# B&R Automation Studio project Ampel
Automation Studio 6.3.2.2; Traffic Ligh in B&R 6.3; technology packages: mappView 6.0.0, OpcUaCs 6.0.0

## Configuration Config1

CPU PC_any, AutomationRuntime 6.3.0, Build 11.3.0, Vc 6.0.0

### Hardware
```
PC : PC_any v1.1.2.0 (OrderNumber=PC)
  ConfigurationID = Ampel_Config1
  FileDevice1
  FileDeviceName1 = USER
  FileDevicePath1 = USER_PATH
```

## Logical view

### Program Logical/Ampel (ANSIC)

#### Main.cpp - Init, cyclic, exit code
```cpp
#include <bur/plctypes.h>

#ifdef _DEFAULT_INCLUDES
#include <AsDefault.h>
#endif

// amount of memory to be allocated for heap storage must be specified
// for every ANSI C++ program with the bur_heap_size variable
unsigned long bur_heap_size = 0xFFFF;

#include "machine.hpp"
#include "Logging.hpp"
#include "States.hpp"

////////////////////////////////////////////////////////////////////////////////

// shared data storage instance
Context context;
FSM::Instance machine{context};

void _INIT ProgramInit(void)
{
	// Insert code here
	CyclesCount = 0;
	ClearTraceLog();
	DurationRed = 5;
	DurationYellow = 3;
	DurationGreen = 5;
	DurationGreenBlinking = 3;
	LightRed = false;
	LightYellow = false;
	LightGreen = false;
	CountDownRedON = false;
	CountDownGreenON = false;
}

void _CYCLIC ProgramCyclic(void)
{
	// Insert code here
	machine.update();
	LightRedOFF = !LightRed; LightYellowOFF = !LightYellow; LightGreenOFF = !LightGreen;
	CountDownRedON = LightRed;
	CyclesCount++;
	TraceMessage("---cycle---");
}

void _EXIT ProgramExit(void)
{
	// Insert code here
}
```

#### Variables.var - Local variables
```iecst
VAR
	DurationGreenBlinking : USINT;
	DurationGreen : USINT;
	DurationYellow : USINT;
	DurationRed : USINT;
	LightYellow : BOOL;
	LightRed : BOOL;
	LightGreen : BOOL;
	CyclesCount : USINT;
	TraceMessages : ARRAY[0..200] OF STRING[80];
	LightYellowOFF : BOOL;
	CountDown : USINT;
	LightRedOFF : BOOL;
	LightGreenOFF : BOOL;
	CountDownRedON : BOOL;
	CountDownGreenON : BOOL;
END_VAR

VAR CONSTANT

END_VAR
```

#### machine.hpp
```cpp
// https://github.com/andrew-gresyk/HFSM2
// include/hfsm2/machine.hpp
// HFSM2 (hierarchical state machine for games and interactive applications)
// 2.8.0 (2025-07-20)
//
// Created by Andrew Gresyk
//
// Licensed under the MIT License;
// you may not use this file except in compliance with the License.
//
//
// MIT License
//
// Copyright (c) 2025
//
// Permission is hereby granted, free of charge, to any person obtaining a copy
// of this software and associated documentation files (the "Software"), to deal
// in the Software without restriction, including without limitation the rights
// to use, copy, modify, merge, publish, distribute, sublicense, and/or sell
// copies of the Software, and to permit persons to whom the Software is
// furnished to do so, subject to the following conditions:
//
// The above copyright notice and this permission notice shall be included in all
// copies or substantial portions of the Software.
//
// THE SOFTWARE IS PROVIDED "AS IS", WITHOUT WARRANTY OF ANY KIND, EXPRESS OR
// IMPLIED, INCLUDING BUT NOT LIMITED TO THE WARRANTIES OF MERCHANTABILITY,
// FITNESS FOR A PARTICULAR PURPOSE AND NONINFRINGEMENT. IN NO EVENT SHALL THE
// AUTHORS OR COPYRIGHT HOLDERS BE LIABLE FOR ANY CLAIM, DAMAGES OR OTHER
// LIABILITY, WHETHER IN AN ACTION OF CONTRACT, TORT OR OTHERWISE, ARISING FROM,
// OUT OF OR IN CONNECTION WITH THE SOFTWARE OR THE USE OR OTHER DEALINGS IN THE
// SOFTWARE.

#pragma once

#define HFSM2_VERSION_MAJOR 2
#define HFSM2_VERSION_MINOR 8
#define HFSM2_VERSION_PATCH 0

#define HFSM2_VERSION (10000 * HFSM2_VERSION_MAJOR + 100 * HFSM2_VERSION_MINOR + HFSM2_VERSION_PATCH)

#include <stdint.h>			// uint32_t, uint64_t
#include <string.h>			// memcpy_s()

#include <new>
#ifndef HFSM2_DISABLE_TYPEINDEX
#include <typeindex>
#endif

#if defined _DEBUG && _MSC_VER
#include <intrin.h>		// __debugbreak()
#endif

#define HFSM2_UNUSED(x)

#define HFSM2_ATTRIBUTE(A)								   HFSM2_ATTRIBUTE_##A()

#ifndef __has_cpp_attribute
#define __has_cpp_attribute(x)											   0
#endif

#if __has_cpp_attribute(fallthrough)
#define HFSM2_ATTRIBUTE_FALLTHROUGH()						 [[fallthrough]]
#elif __has_cpp_attribute(clang::fallthrough)
#define HFSM2_ATTRIBUTE_FALLTHROUGH()				  [[clang::fallthrough]]
#elif __has_cpp_attribute(gnu::fallthrough)
#define HFSM2_ATTRIBUTE_FALLTHROUGH()					[[gnu::fallthrough]]
#else
#define HFSM2_ATTRIBUTE_FALLTHROUGH()
#endif

#if __has_cpp_attribute(no_unique_address)
#define HFSM2_ATTRIBUTE_NO_UNIQUE_ADDRESS()			   [[no_unique_address]]
#else
#define HFSM2_ATTRIBUTE_NO_UNIQUE_ADDRESS()
#endif

#define HFSM2_CONSTEXPR(A)								   HFSM2_CONSTEXPR_##A()

#define HFSM2_CONSTEXPR_NO()

#define HFSM2_CONSTEXPR_11()										   constexpr

#if __cplusplus >= 201402L
#define HFSM2_CONSTEXPR_14()									   constexpr
#else
#define HFSM2_CONSTEXPR_14()										  inline
#endif

#if __cplusplus >= 201703L
#define HFSM2_CONSTEXPR_17()									   constexpr
#else
#define HFSM2_CONSTEXPR_17()										  inline
#endif

#if __cplusplus >= 202002L
#define HFSM2_CONSTEXPR_20()									   constexpr
#else
#define HFSM2_CONSTEXPR_20()										  inline
#endif

#if defined _MSC_VER
#define HFSM2_EMPTY_BASES							 __declspec(empty_bases)
#else
#define HFSM2_EMPTY_BASES
#endif

#define HFSM2_ARCHITECTURE(A)							HFSM2_ARCHITECTURE_##A()

#if INTPTR_MAX == INT64_MAX
#define HFSM2_ARCHITECTURE_64BIT()										true
#define HFSM2_ARCHITECTURE_32BIT()									   false

#define HFSM2_64BIT_OR_32BIT(p64, p32)									 p64
#elif INTPTR_MAX == INT32_MAX
#define HFSM2_ARCHITECTURE_64BIT()									   false
#define HFSM2_ARCHITECTURE_32BIT()										true

#define HFSM2_64BIT_OR_32BIT(p64, p32)									 p32
#else
#error
#endif

#if defined _DEBUG && defined _MSC_VER
#define HFSM2_BREAK()										  __debugbreak()
#define HFSM2_BREAK_AVAILABLE()											true
#else
#define HFSM2_BREAK()											  ((void) 0)
#define HFSM2_BREAK_AVAILABLE()										   false
#endif

#ifdef _DEBUG
#define HFSM2_IF_DEBUG(...)										 __VA_ARGS__
#define HFSM2_UNLESS_DEBUG(...)
#define HFSM2_DEBUG_OR(y, n)											   y
#else
#define HFSM2_IF_DEBUG(...)
#define HFSM2_UNLESS_DEBUG(...)									 __VA_ARGS__
#define HFSM2_DEBUG_OR(y, n)											   n
#endif

#if HFSM2_BREAK_AVAILABLE() && defined HFSM2_ENABLE_ASSERT
#define HFSM2_ASSERT_AVAILABLE()										true
#define HFSM2_IF_ASSERT(...)									 __VA_ARGS__
#define HFSM2_CHECKED(x)					   (!!(x) || (HFSM2_BREAK(), 0))
#define HFSM2_ASSERT(x)						   (!!(x) || (HFSM2_BREAK(), 0))
#define HFSM2_ASSERT_OR(y, n)											   y
#else
#define HFSM2_ASSERT_AVAILABLE()									   false
#define HFSM2_IF_ASSERT(...)
#define HFSM2_CHECKED(x)												   x
#define HFSM2_ASSERT(x)											  ((void) 0)
#define HFSM2_ASSERT_OR(y, n)											   n
#endif

#if defined _MSC_VER || defined __clang_major__ && __clang_major__ >= 7
#define HFSM2_EXPLICIT_MEMBER_SPECIALIZATION_AVAILABLE()				true
#else
#define HFSM2_EXPLICIT_MEMBER_SPECIALIZATION_AVAILABLE()			   false
#endif

#ifdef HFSM2_ENABLE_ALL
#define HFSM2_ENABLE_DEBUG_STATE_TYPE
#define HFSM2_ENABLE_PLANS
#define HFSM2_ENABLE_SERIALIZATION
#define HFSM2_ENABLE_STRUCTURE_REPORT
#define HFSM2_ENABLE_TRANSITION_HISTORY
#define HFSM2_ENABLE_UTILITY_THEORY
#endif

#ifndef HFSM2_DISABLE_TYPEINDEX
#define HFSM2_TYPEINDEX_AVAILABLE()										true
#define HFSM2_IF_TYPEINDEX(...)									 __VA_ARGS__
#define HFSM2_TYPEINDEX_MASK										(1 << 0)
#else
#define HFSM2_TYPEINDEX_AVAILABLE()									   false
#define HFSM2_IF_TYPEINDEX(...)
#define HFSM2_TYPEINDEX_MASK										(0 << 0)
#endif

#ifdef HFSM2_ENABLE_DEBUG_STATE_TYPE
#define HFSM2_DEBUG_STATE_TYPE_AVAILABLE()								true
#define HFSM2_DEBUG_STATE_TYPE_MASK									(1 << 1)
#else
#define HFSM2_DEBUG_STATE_TYPE_AVAILABLE()							   false
#define HFSM2_DEBUG_STATE_TYPE_MASK									(0 << 1)
#endif

#ifdef HFSM2_ENABLE_PLANS
#define HFSM2_PLANS_AVAILABLE()											true
#define HFSM2_IF_PLANS(...)										 __VA_ARGS__
#define HFSM2_PLANS_MASK											(1 << 2)
#else
#define HFSM2_PLANS_AVAILABLE()										   false
#define HFSM2_IF_PLANS(...)
#define HFSM2_PLANS_MASK											(0 << 2)
#endif

#ifdef HFSM2_ENABLE_SERIALIZATION
#define HFSM2_SERIALIZATION_AVAILABLE()									true
#define HFSM2_IF_SERIALIZATION(...)								 __VA_ARGS__
#define HFSM2_SERIALIZATION_MASK									(1 << 3)
#else
#define HFSM2_SERIALIZATION_AVAILABLE()								   false
#define HFSM2_IF_SERIALIZATION(...)
#define HFSM2_SERIALIZATION_MASK									(0 << 3)
#endif

#ifdef HFSM2_ENABLE_STRUCTURE_REPORT
#define HFSM2_STRUCTURE_REPORT_AVAILABLE()								true
#define HFSM2_IF_STRUCTURE_REPORT(...)							 __VA_ARGS__
#define HFSM2_STRUCTURE_REPORT_MASK									(1 << 4)
#else
#define HFSM2_STRUCTURE_REPORT_AVAILABLE()							   false
#define HFSM2_IF_STRUCTURE_REPORT(...)
#define HFSM2_STRUCTURE_REPORT_MASK									(0 << 4)
#endif

#ifdef HFSM2_ENABLE_TRANSITION_HISTORY
#define HFSM2_TRANSITION_HISTORY_AVAILABLE()							true
#define HFSM2_IF_TRANSITION_HISTORY(...)						 __VA_ARGS__
#define HFSM2_TRANSITION_HISTORY_MASK								(1 << 5)
#else
#define HFSM2_TRANSITION_HISTORY_AVAILABLE()						   false
#define HFSM2_IF_TRANSITION_HISTORY(...)
#define HFSM2_TRANSITION_HISTORY_MASK								(0 << 5)
#endif

#ifdef HFSM2_ENABLE_UTILITY_THEORY
#define HFSM2_UTILITY_THEORY_AVAILABLE()								true
#define HFSM2_IF_UTILITY_THEORY(...)							 __VA_ARGS__
#define HFSM2_UTILITY_THEORY_MASK									(1 << 6)
#else
#define HFSM2_UTILITY_THEORY_AVAILABLE()							   false
#define HFSM2_IF_UTILITY_THEORY(...)
#define HFSM2_UTILITY_THEORY_MASK									(0 << 6)
#endif

#ifdef HFSM2_ENABLE_VERBOSE_DEBUG_LOG
#define HFSM2_ENABLE_LOG_INTERFACE

#define HFSM2_VERBOSE_DEBUG_LOG_AVAILABLE()								true
#define HFSM2_VERBOSE_DEBUG_LOG_MASK								(1 << 7)
#else
#define HFSM2_VERBOSE_DEBUG_LOG_AVAILABLE()							   false
#define HFSM2_VERBOSE_DEBUG_LOG_MASK								(0 << 7)
#endif

#ifdef HFSM2_ENABLE_LOG_INTERFACE
#define HFSM2_LOG_INTERFACE_AVAILABLE()									true
#define HFSM2_IF_LOG_INTERFACE(...)								 __VA_ARGS__
#define HFSM2_LOG_INTERFACE_MASK									(1 << 8)

#define HFSM2_LOG_TRANSITION(CONTEXT, ORIGIN, TYPE, DESTINATION)		   \
		if (_core.logger)													   \
			_core.logger->recordTransition(CONTEXT, ORIGIN, TYPE, DESTINATION)

#if HFSM2_PLANS_AVAILABLE()
#define HFSM2_LOG_TASK_STATUS(CONTEXT, REGION, ORIGIN, STATUS)			   \
		if (_core.logger)													   \
			_core.logger->recordTaskStatus(CONTEXT, REGION, ORIGIN, STATUS)

#define HFSM2_LOG_PLAN_STATUS(CONTEXT, REGION, STATUS)					   \
		if (_core.logger)													   \
			_core.logger->recordPlanStatus(CONTEXT, REGION, STATUS)
#endif

#define HFSM2_LOG_CANCELLED_PENDING(CONTEXT, ORIGIN)					   \
		if (_core.logger)													   \
			_core.logger->recordCancelledPending(CONTEXT, ORIGIN)

#define HFSM2_LOG_SELECT_RESOLUTION(CONTEXT, HEAD, PRONG)				   \
		if (auto* const logger = control._core.logger)						   \
			logger->recordSelectResolution(CONTEXT, HEAD, PRONG)

#if HFSM2_UTILITY_THEORY_AVAILABLE()
#define HFSM2_LOG_UTILITY_RESOLUTION(CONTEXT, HEAD, PRONG, UTILITY)		   \
		if (auto* const logger = control._core.logger)						   \
			logger->recordUtilityResolution(CONTEXT, HEAD, PRONG, UTILITY)

#define HFSM2_LOG_RANDOM_RESOLUTION(CONTEXT, HEAD, PRONG, UTILITY)		   \
		if (auto* const logger = control._core.logger)						   \
			logger->recordRandomResolution(CONTEXT, HEAD, PRONG, UTILITY)
#endif

#else

#define HFSM2_LOG_INTERFACE_AVAILABLE()								   false
#define HFSM2_IF_LOG_INTERFACE(...)
#define HFSM2_LOG_INTERFACE_MASK									(0 << 8)

#define HFSM2_LOG_TRANSITION(CONTEXT, ORIGIN, TYPE, DESTINATION)

#if HFSM2_PLANS_AVAILABLE()
#define HFSM2_LOG_TASK_STATUS(CONTEXT, REGION, ORIGIN, STATUS)
#define HFSM2_LOG_PLAN_STATUS(CONTEXT, REGION, STATUS)
#endif

#define HFSM2_LOG_CANCELLED_PENDING(CONTEXT, ORIGIN)
#define HFSM2_LOG_SELECT_RESOLUTION(CONTEXT, HEAD, PRONG)

#if HFSM2_UTILITY_THEORY_AVAILABLE()
#define HFSM2_LOG_UTILITY_RESOLUTION(CONTEXT, HEAD, PRONG, UTILITY)
#define HFSM2_LOG_RANDOM_RESOLUTION(CONTEXT, HEAD, PRONG, UTILITY)
#endif

#endif

#if HFSM2_VERBOSE_DEBUG_LOG_AVAILABLE()

#define HFSM2_LOG_STATE_METHOD(METHOD, METHOD_ID)						   \
		if (auto* const logger = control._core.logger)						   \
			logger->recordMethod(control.context(), STATE_ID, METHOD_ID)

#define HFSM2_IF_LOG_STATE_METHOD(...)							 __VA_ARGS__
#define HFSM2_IF_PLANS_OR_LOG_STATE_METHOD(...)					 __VA_ARGS__

#elif HFSM2_LOG_INTERFACE_AVAILABLE()

#define HFSM2_LOG_STATE_METHOD(METHOD, METHOD_ID)						   \
		if (auto* const logger = control._core.logger)						   \
			log(METHOD, *logger, control.context(), METHOD_ID)

#define HFSM2_IF_LOG_STATE_METHOD(...)							 __VA_ARGS__
#define HFSM2_IF_PLANS_OR_LOG_STATE_METHOD(...)					 __VA_ARGS__

#else

#define HFSM2_LOG_STATE_METHOD(METHOD, METHOD_ID)

#define HFSM2_IF_LOG_STATE_METHOD(...)

#if HFSM2_PLANS_AVAILABLE()
#define HFSM2_IF_PLANS_OR_LOG_STATE_METHOD(...)				 __VA_ARGS__
#else
#define HFSM2_IF_PLANS_OR_LOG_STATE_METHOD(...)
#endif

#endif

namespace hfsm2 {

	using FeatureTag = uint16_t;

	constexpr FeatureTag HFSM2_FEATURE_TAG = HFSM2_TYPEINDEX_MASK
		| HFSM2_DEBUG_STATE_TYPE_MASK
		| HFSM2_PLANS_MASK
		| HFSM2_SERIALIZATION_MASK
		| HFSM2_STRUCTURE_REPORT_MASK
		| HFSM2_TRANSITION_HISTORY_MASK
		| HFSM2_UTILITY_THEORY_MASK
		| HFSM2_VERBOSE_DEBUG_LOG_MASK
		| HFSM2_LOG_INTERFACE_MASK;

}

#undef HFSM2_TYPEINDEX_MASK
#undef HFSM2_DEBUG_STATE_TYPE_MASK
#undef HFSM2_PLANS_MASK
#undef HFSM2_SERIALIZATION_MASK
#undef HFSM2_STRUCTURE_REPORT_MASK
#undef HFSM2_TRANSITION_HISTORY_MASK
#undef HFSM2_UTILITY_THEORY_MASK
#undef HFSM2_VERBOSE_DEBUG_LOG_MASK
#undef HFSM2_LOG_INTERFACE_MASK

#if _MSC_VER == 1900
#pragma warning(push)
#pragma warning(disable: 4814) // in C++14 'constexpr' will not imply 'const'; consider explicitly specifying 'const'
#endif

#ifdef __clang__
#pragma clang diagnostic push
#pragma clang diagnostic ignored "-Wextra-semi" // error : extra ';' inside a class
#pragma clang diagnostic ignored "-Wconstexpr-not-const" // error: 'constexpr' non-static member function will not be implicitly 'const' in C++14; add 'const' to avoid a change in behavior
#endif

#if defined(__GNUC__) || defined(__GNUG__)
#pragma GCC diagnostic push
#pragma GCC diagnostic ignored "-Wpedantic" // error : extra ';'
#endif

namespace hfsm2 {

	struct EmptyPayload final {};

struct Automatic;
struct Manual;

struct TopDown;
struct BottomUp;

using Short		 = uint8_t;
static constexpr Short		INVALID_SHORT		= UINT8_MAX;

using Long		 = uint16_t;
static constexpr Long		INVALID_LONG		= UINT16_MAX;

using Prong		 = Short;
static constexpr Prong		INVALID_PRONG		= INVALID_SHORT;

using RegionID	 = Short;
static constexpr RegionID	INVALID_REGION_ID	= INVALID_SHORT;

using ForkID	 = int16_t;
static constexpr ForkID		INVALID_FORK_ID		= INT16_MIN;

using StateID	 = Long;
static constexpr StateID	INVALID_STATE_ID	= INVALID_LONG;
static constexpr StateID	ROOT_ID				= 0;

template <
	bool B
  , typename TT
  , typename TF
>
struct ConditionalT final {
	using Type = TT;
};

template <
	typename TT
  , typename TF
>
struct ConditionalT<false, TT, TF> final {
	using Type = TF;
};

template <
	bool B
  , typename TT
  , typename TF
>
using Conditional = typename ConditionalT<B, TT, TF>::Type;

template <typename T>
struct RemoveConstT final {
	using Type = T;
};

template <typename T>
struct RemoveConstT<const T> final {
	using Type = T;
};

template <typename T>
using RemoveConst = typename RemoveConstT<T>::Type;

template <typename T>
struct RemoveReferenceT final {
	using Type = T;
};

template <typename T>
struct RemoveReferenceT<T&> final {
	using Type = T;
};

template <typename T>
struct RemoveReferenceT<T&&> final {
	using Type = T;
};

template <typename T>
using RemoveReference = typename RemoveReferenceT<T>::Type;

template <typename T>
using Undecorate = RemoveConst<RemoveReference<T>>;

template <typename T>
struct IsValueReferenceT final {
	static const bool VALUE = false;
};

template <typename T>
struct IsValueReferenceT<T&> final {
	static const bool VALUE = true;
};

template <uint64_t N>
using UIndex = Conditional<N <= (1ull <<  8),  uint8_t,
			   Conditional<N <= (1ull << 16), uint16_t,
			   Conditional<N <= (1ull << 32), uint32_t,
												  void>>>;

template <uint64_t N>
using UCapacity = Conditional<N < (1ull <<  8),  uint8_t,
	Conditional<N < (1ull << 16), uint16_t,
	Conditional<N < (1ull << 32), uint32_t,
	void>>>;

HFSM2_CONSTEXPR(11)
Short
bitContain(const Short v)												noexcept	{
	return v <= 1 << 0 ? 0 :
		   v <= 1 << 1 ? 1 :
		   v <= 1 << 2 ? 2 :
		   v <= 1 << 3 ? 3 :
		   v <= 1 << 4 ? 4 :
		   v <= 1 << 5 ? 5 :
		   v <= 1 << 6 ? 6 :
		   v <= 1 << 7 ? 7 :
						 8 ;
}

template <uint64_t N>
using UBitWidth = Conditional<N <=  8,  uint8_t,
	Conditional<N <= 16, uint16_t,
	Conditional<N <= 32, uint32_t,
	void>>>;

template <typename T>
HFSM2_CONSTEXPR(11)
T&&
forward(RemoveReference<T>& t)											noexcept	{
	return static_cast<T&&>(t);
}

template <typename T>
HFSM2_CONSTEXPR(11)
T&&
forward(RemoveReference<T>&& t)											noexcept	{
	static_assert(!IsValueReferenceT<T>::VALUE, "");

	return static_cast<T&&>(t);
}

template <typename T>
HFSM2_CONSTEXPR(11)
RemoveReference<T>&&
move(T&& t)																noexcept	{
	return static_cast<RemoveReference<T>&&>(t);
}

template <
	typename T0
  , typename T1
>
HFSM2_CONSTEXPR(11)
T0
min(const T0 t0,
	const T1 t1)														noexcept
{
	return t0 < static_cast<T0>(t1) ?
		   t0 : static_cast<T0>(t1);
}

template <
	typename T0
  , typename T1
>
HFSM2_CONSTEXPR(11)
T0
max(const T0 t0,
	const T1 t1)														noexcept
{
	return t0 > static_cast<T0>(t1) ?
		   t0 : static_cast<T0>(t1);
}

template <
	typename TIndex
  , typename TElement
  , TIndex NCount
>
HFSM2_CONSTEXPR(11)
TIndex
count(const TElement (&)[NCount])										noexcept	{
return NCount;
}

template <
	typename T
  , typename TT
>
HFSM2_CONSTEXPR(11)
T
contain(const T x,
		const TT to)													noexcept
{
	return (x + static_cast<T>(to) - 1) / static_cast<T>(to);
}

HFSM2_CONSTEXPR(11)
uint64_t
widen(const uint32_t x, const uint32_t y)								noexcept	{
return static_cast<uint64_t>(x) << 32 | y;
}

template <typename T>
HFSM2_CONSTEXPR(14)
void
fill(T& a, const char value)											noexcept	{
	memset(&a, static_cast<int>(value), sizeof(a));
}

template <typename T>
HFSM2_CONSTEXPR(14)
void
swap(T& l, T& r)														noexcept	{
T t = move(l);
l = move(r);
r = move(t);
}

template <
	typename TTo
  , typename TFrom
>
HFSM2_CONSTEXPR(14)
void
overwrite(TTo& to, const TFrom& from)									noexcept	{
	static_assert(sizeof(TTo) == sizeof(TFrom), "");

#if defined(__GNUC__) || defined(__GNUG__)
	memcpy  (&to,			  &from, sizeof(from));
#else
	memcpy_s(&to, sizeof(to), &from, sizeof(from));
#endif
}

template <
	typename TO
  , typename TI
>
HFSM2_CONSTEXPR(14)
TO
reinterpret(const TI& in)												noexcept	{
TO out{};

	overwrite(out, in);

return out;
}

template<class T>
HFSM2_CONSTEXPR(14)
void destroy(T& t)														noexcept	{
	t.~T();
}

template <int>
struct StaticPrintConstT;

template <typename>
struct StaticPrintTypeT;

}

namespace hfsm2 {
	namespace detail {

		template <typename TContainer>
		class IteratorT {
			public:
			using Container = TContainer;
			using Item		= typename Container::Item;
			using Index		= typename Container::Index;

			template <typename, Long>
			friend class DynamicArrayT;

			private:
			HFSM2_CONSTEXPR(11)	IteratorT(Container& container,
			const Index cursor)										noexcept
		: _container{container}
	, _cursor{cursor}
{}

public:
	HFSM2_CONSTEXPR(14)	bool operator != (const IteratorT& HFSM2_IF_ASSERT(other))	  const noexcept	{
		HFSM2_ASSERT(&_container == &other._container);

		return _cursor != _container.limit();
	}

	HFSM2_CONSTEXPR(14)	IteratorT& operator ++()											noexcept	{
	_cursor = _container.next(_cursor);

	return *this;
}

	HFSM2_CONSTEXPR(14)		  Item& operator *()			noexcept	{ return  _container[_cursor];	}
	HFSM2_CONSTEXPR(11)	const Item& operator *()	  const noexcept	{ return  _container[_cursor];	}

	HFSM2_CONSTEXPR(14)		  Item* operator->()			noexcept	{ return &_container[_cursor];	}
	HFSM2_CONSTEXPR(11)	const Item* operator->()	  const noexcept	{ return &_container[_cursor];	}

private:
Container& _container;

Index _cursor;
};

template <typename TContainer>
class IteratorT<const TContainer> {
	public:
	using Container = TContainer;
	using Item		= typename Container::Item;
	using Index		= typename Container::Index;

	template <typename, Long>
	friend class DynamicArrayT;

	private:
	HFSM2_CONSTEXPR(11)	IteratorT(const Container& container,
	const Index cursor)										noexcept
: _container{container}
		, _cursor{cursor}
	{}

public:
	HFSM2_CONSTEXPR(14)	bool operator != (const IteratorT& HFSM2_IF_ASSERT(other))	  const noexcept	{
		HFSM2_ASSERT(&_container == &other._container);

		return _cursor != _container.limit();
	}

	HFSM2_CONSTEXPR(14)	IteratorT& operator ++()											noexcept	{
	_cursor = _container.next(_cursor);

	return *this;
}

	HFSM2_CONSTEXPR(11)	const Item& operator *()	  const noexcept	{ return _container[_cursor];	}

	HFSM2_CONSTEXPR(11)	const Item* operator->()	  const noexcept	{ return &operator *();			}

private:
const Container& _container;

Index _cursor;
};

}
}

#if HFSM2_SERIALIZATION_AVAILABLE()

namespace hfsm2 {
	namespace detail {

		template <Long>
		class BitWriteStreamT;

		template <Long>
		class BitReadStreamT;

		template <Long NBitCapacity>
		class StreamBufferT {
			template <Long>
			friend class BitWriteStreamT;

			template <Long>
			friend class BitReadStreamT;

			public:
			static constexpr Long BIT_CAPACITY	= NBitCapacity;
			static constexpr Long BYTE_COUNT	= contain(BIT_CAPACITY, 8u);

			using StreamBuffer	= StreamBufferT<BIT_CAPACITY>;
			using Data			= uint8_t	   [BYTE_COUNT	];

		HFSM2_CONSTEXPR(14)	void clear()									noexcept	{ fill(_data, 0);	}

	HFSM2_CONSTEXPR(14)		  Data& data()								noexcept	{ return _data;		}
	HFSM2_CONSTEXPR(11)	const Data& data()						  const noexcept	{ return _data;		}

	HFSM2_CONSTEXPR(14) bool operator == (const StreamBuffer& s)  const noexcept;
	HFSM2_CONSTEXPR(14) bool operator != (const StreamBuffer& s)  const noexcept;

	private:
	Data _data {};
};

template <Long NBitCapacity>
class BitWriteStreamT final {
	public:
	static constexpr Long BIT_CAPACITY = NBitCapacity;

	using Buffer = StreamBufferT<BIT_CAPACITY>;

	public:
	HFSM2_CONSTEXPR(14)	explicit BitWriteStreamT(Buffer& buffer,
	const Long cursor = 0)	noexcept
: _buffer{buffer}
		, _cursor{cursor}
	{
		_buffer.clear();
	}

	template <Short NBitWidth>
	HFSM2_CONSTEXPR(14)	void write(const UBitWidth<NBitWidth> item)		noexcept;

	HFSM2_CONSTEXPR(11)	Long cursor()							  const noexcept	{ return _cursor;	}

private:
Buffer& _buffer;

Long _cursor = 0;
};

template <Long NBitCapacity>
class BitReadStreamT final {
	public:
	static constexpr Long BIT_CAPACITY = NBitCapacity;

	using Buffer = StreamBufferT<BIT_CAPACITY>;

	public:
	HFSM2_CONSTEXPR(11)	explicit BitReadStreamT(const Buffer& buffer,
	const Long cursor = 0)	noexcept
: _buffer{buffer}
		, _cursor{cursor}
	{}

	template <Short NBitWidth>
	HFSM2_CONSTEXPR(14)	UBitWidth<NBitWidth> read()						noexcept;

	HFSM2_CONSTEXPR(11)	Long cursor()							  const noexcept	{ return _cursor;	}

private:
const Buffer& _buffer;

Long _cursor;
};

}
}

#if HFSM2_SERIALIZATION_AVAILABLE()

namespace hfsm2 {
namespace detail {

template <Long NBitCapacity>
HFSM2_CONSTEXPR(14)
bool
StreamBufferT<NBitCapacity>::operator == (const StreamBuffer& buffer) const noexcept {
	for (Long i = 0; i < BYTE_COUNT; ++i)
		if (_data[i] != buffer._data[i])
			return false;

	return true;
}

template <Long NBitCapacity>
HFSM2_CONSTEXPR(14)
bool
StreamBufferT<NBitCapacity>::operator != (const StreamBuffer& buffer) const noexcept {
	for (Long i = 0; i < BYTE_COUNT; ++i)
		if (_data[i] != buffer._data[i])
			return true;

	return false;
}

template <Long NBitCapacity>
template <Short NBitWidth>
HFSM2_CONSTEXPR(14)
void
BitWriteStreamT<NBitCapacity>::write(const UBitWidth<NBitWidth> item) noexcept {
constexpr Short BIT_WIDTH = NBitWidth;
	static_assert(BIT_WIDTH > 0, "STATIC ASSERT");

	HFSM2_ASSERT(_cursor + BIT_WIDTH <= BIT_CAPACITY);

	using Item = UBitWidth<BIT_WIDTH>;

Item itemBits = item;

for (Short itemWidth = BIT_WIDTH; itemWidth; ) {
const Long	byteIndex		= _cursor >> 3;
uint8_t&	byte			= _buffer._data[byteIndex];

const Short byteChunkStart	= _cursor & 0x7;
const Short byteDataWidth	= 8 - byteChunkStart;
const Short byteChunkWidth	= min(byteDataWidth, itemWidth);
const Item	byteChunk		= itemBits << byteChunkStart;

byte		|= byteChunk;
itemBits   >>= byteChunkWidth;
itemWidth	-= byteChunkWidth;
_cursor		+= byteChunkWidth;
	}
}

template <Long NBitCapacity>
template <Short NBitWidth>
HFSM2_CONSTEXPR(14)
UBitWidth<NBitWidth>
BitReadStreamT<NBitCapacity>::read() noexcept {
constexpr Short BIT_WIDTH = NBitWidth;
	static_assert(BIT_WIDTH > 0, "STATIC ASSERT");

	HFSM2_ASSERT(_cursor + BIT_WIDTH <= BIT_CAPACITY);

	using Item = UBitWidth<BIT_WIDTH>;

Item item = 0;

for (Short itemCursor = 0, itemWidth = BIT_WIDTH; itemWidth; ) {
const Long	byteIndex		= _cursor >> 3;
const uint8_t& byte			= _buffer._data[byteIndex];

const Short byteChunkStart	= _cursor & 0x7;
const Short byteDataWidth	= 8 - byteChunkStart;
const Short byteChunkWidth	= min(byteDataWidth, itemWidth);
const Short byteChunkMask	= (1 << byteChunkWidth) - 1;

const Item	byteChunk		= (byte >> byteChunkStart) & byteChunkMask;
const Item	itemChunk		= byteChunk << itemCursor;

item		|= itemChunk;
itemCursor	+= byteChunkWidth;
itemWidth	-= byteChunkWidth;
_cursor		+= byteChunkWidth;
	}

return item;
}

}
}

#endif

#endif

#if HFSM2_UTILITY_THEORY_AVAILABLE()

namespace hfsm2 {
	namespace detail {

		HFSM2_CONSTEXPR(14)	float  uniform(const uint32_t uint)					noexcept;
		HFSM2_CONSTEXPR(14)	double uniform(const uint64_t uint)					noexcept;

		template <unsigned>
		struct SimpleRandomT;

// SplitMix64 (http://xoshiro.di.unimi.it/splitmix64.c)

		template <>
		struct SimpleRandomT<8> {
		HFSM2_CONSTEXPR(11) SimpleRandomT()									noexcept	{}
		HFSM2_CONSTEXPR(14)	SimpleRandomT(const uint64_t seed)				noexcept;

		HFSM2_CONSTEXPR(14)	uint64_t uint64()								noexcept;
		HFSM2_CONSTEXPR(14)	uint64_t raw64()								noexcept;

		uint64_t _state = 0;
	};

// SplitMix32 (https://groups.google.com/forum/#!topic/prng/VFjdFmbMgZI)

	template <>
	struct SimpleRandomT<4> {
	HFSM2_CONSTEXPR(11)	SimpleRandomT()									noexcept	{}
	HFSM2_CONSTEXPR(14)	SimpleRandomT(const uint32_t seed)				noexcept;

	HFSM2_CONSTEXPR(14)	uint32_t uint32()								noexcept;
	HFSM2_CONSTEXPR(14)	uint32_t raw32()								noexcept;

	uint32_t _state = 0;
};

template <unsigned>
class BaseRandomT;

template <>
class BaseRandomT<8> {
	protected:
	using SimpleRandom = SimpleRandomT<8>;

	HFSM2_CONSTEXPR(14)	BaseRandomT(SimpleRandom&& simple)				noexcept;

	HFSM2_CONSTEXPR(14)	void seed(SimpleRandom&& simple)				noexcept;

	public:
	HFSM2_CONSTEXPR(14)	BaseRandomT()									noexcept;

	HFSM2_CONSTEXPR(14)	BaseRandomT(const uint64_t s)					noexcept;
	HFSM2_CONSTEXPR(14)	BaseRandomT(const uint64_t(& s)[4])				noexcept;

	HFSM2_CONSTEXPR(14)	void seed(const uint64_t s)						noexcept;
	HFSM2_CONSTEXPR(14)	void seed(const uint64_t(& s)[4])				noexcept;

	protected:
	uint64_t _state[4] {};
};

template <>
class BaseRandomT<4> {
	protected:
	using SimpleRandom = SimpleRandomT<4>;

	HFSM2_CONSTEXPR(14)	BaseRandomT(SimpleRandom&& simple)				noexcept;

	HFSM2_CONSTEXPR(14)	void seed(SimpleRandom&& simple)				noexcept;

	public:
	HFSM2_CONSTEXPR(14)	BaseRandomT()									noexcept;

	HFSM2_CONSTEXPR(14)	BaseRandomT(const uint32_t s)					noexcept;
	HFSM2_CONSTEXPR(14)	BaseRandomT(const uint32_t(& s)[4])				noexcept;

	HFSM2_CONSTEXPR(14)	void seed(const uint32_t s)						noexcept;
	HFSM2_CONSTEXPR(14)	void seed(const uint32_t(& s)[4])				noexcept;

	protected:
	uint32_t _state[4] {};
};

template <unsigned>
class FloatRandomT;

// xoshiro256+ (http://xoshiro.di.unimi.it/xoshiro256plus.c)

template <>
class FloatRandomT<8>
	: BaseRandomT<8>
	{
	using Base = BaseRandomT<8>;

	public:
	using Base::BaseRandomT;

HFSM2_CONSTEXPR(14)	double	float64()								noexcept	{ return uniform(uint64());					}
	HFSM2_CONSTEXPR(14)	float	float32()								noexcept	{ return uniform(uint32());					}

	HFSM2_CONSTEXPR(14)	uint64_t uint64()								noexcept;
	HFSM2_CONSTEXPR(14)	uint32_t uint32()								noexcept	{ return static_cast<uint32_t>(uint64());	}

	HFSM2_CONSTEXPR(14)	float next()									noexcept	{ return float32();							}
	HFSM2_CONSTEXPR(14)	void  jump()									noexcept;
};

// xoshiro128+ (http://xoshiro.di.unimi.it/xoshiro128plus.c)

template <>
class FloatRandomT<4>
	: BaseRandomT<4>
	{
	using Base = BaseRandomT<4>;

	public:
	using Base::BaseRandomT;

HFSM2_CONSTEXPR(14)	double	float64()								noexcept	{ return uniform(uint64());					}
	HFSM2_CONSTEXPR(14)	float	float32()								noexcept	{ return uniform(uint32());					}

	HFSM2_CONSTEXPR(14)	uint64_t uint64()								noexcept	{ return widen(uint32(), uint32());			}
	HFSM2_CONSTEXPR(14)	uint32_t uint32()								noexcept;

	HFSM2_CONSTEXPR(14)	float next()									noexcept	{ return float32();							}
	HFSM2_CONSTEXPR(14)	void  jump()									noexcept;
};

template <unsigned>
class IntRandomT;

// xoshiro256** (https://prng.di.unimi.it/xoshiro256starstar.c)

template <>
class IntRandomT<8>
	: BaseRandomT<8>
	{
	using Base = BaseRandomT<8>;

	public:
	using Base::BaseRandomT;

HFSM2_CONSTEXPR(14)	double	float64()								noexcept	{ return uniform(uint64());					}
	HFSM2_CONSTEXPR(14)	float	float32()								noexcept	{ return uniform(uint32());					}

	HFSM2_CONSTEXPR(14)	uint64_t uint64()								noexcept;
	HFSM2_CONSTEXPR(14)	uint32_t uint32()								noexcept	{ return static_cast<uint32_t>(uint64());	}

	HFSM2_CONSTEXPR(14)	void jump()										noexcept;
};

// xoshiro128** (https://prng.di.unimi.it/xoshiro128starstar.c)

template <>
class IntRandomT<4>
	: BaseRandomT<4>
	{
	using Base = BaseRandomT<4>;

	public:
	using Base::BaseRandomT;

HFSM2_CONSTEXPR(14)	double	float64()								noexcept	{ return uniform(uint64());			}
	HFSM2_CONSTEXPR(14)	float	float32()								noexcept	{ return uniform(uint32());			}

	HFSM2_CONSTEXPR(14)	uint64_t uint64()								noexcept	{ return widen(uint32(), uint32());	}
	HFSM2_CONSTEXPR(14)	uint32_t uint32()								noexcept;

	HFSM2_CONSTEXPR(14)	void jump()										noexcept;
};

}

using SimpleRandom = detail::SimpleRandomT<sizeof(void*)>;
using FloatRandom  = detail::FloatRandomT <sizeof(void*)>;
using IntRandom	   = detail::IntRandomT	  <sizeof(void*)>;

template <typename T>
class RNGT;

template <>
class RNGT<float>
	: public FloatRandom
{
	public:
	using Base = FloatRandom;

	using Base::Base;
};

template <>
class RNGT<uintptr_t>
	: public IntRandom
{
	public:
	using Base = IntRandom;

	using Base::Base;
};

}

#endif

#if HFSM2_UTILITY_THEORY_AVAILABLE()

namespace hfsm2 {
namespace detail {

HFSM2_CONSTEXPR(14)
float
uniform(const uint32_t uint) noexcept {
	return reinterpret<float>(UINT32_C(0x7F) << 23 | uint >> 9) - 1.0f;
}

HFSM2_CONSTEXPR(14)
double
uniform(const uint64_t uint) noexcept {
	return reinterpret<double>(UINT64_C(0x3FF) << 52 | uint >> 12) - 1.0;
}

HFSM2_CONSTEXPR(11)
uint32_t
rotl(const uint32_t x, const uint32_t k) noexcept {
	return (x << k) | (x >> (32 - k));
}

HFSM2_CONSTEXPR(11)
uint64_t
rotl(const uint64_t x, const uint64_t k) noexcept {
	return (x << k) | (x >> (64 - k));
}

HFSM2_CONSTEXPR(14)
SimpleRandomT<8>::SimpleRandomT(const uint64_t seed) noexcept
	: _state{seed}
{}

HFSM2_CONSTEXPR(14)
uint64_t
SimpleRandomT<8>::uint64() noexcept {
	for (;;)
if (const uint64_t number = raw64())
return number;
}

HFSM2_CONSTEXPR(14)
uint64_t
SimpleRandomT<8>::raw64() noexcept {
uint64_t z = (_state += 0x9e3779b97f4a7c15);
z = (z ^ (z >> 30)) * 0xbf58476d1ce4e5b9;
z = (z ^ (z >> 27)) * 0x94d049bb133111eb;

	return z ^ (z >> 31);
}

HFSM2_CONSTEXPR(14)
SimpleRandomT<4>::SimpleRandomT(const uint32_t seed) noexcept
	: _state{seed}
{}

HFSM2_CONSTEXPR(14)
uint32_t
SimpleRandomT<4>::uint32() noexcept {
	for (;;)
if (const uint32_t number = raw32())
return number;
}

HFSM2_CONSTEXPR(14)
uint32_t
SimpleRandomT<4>::raw32() noexcept {
uint32_t z = (_state += 0x9E3779B9);
z = (z ^ (z >> 16)) * 0x85ebca6b;
z = (z ^ (z >> 13)) * 0xc2b2ae35;

	return z ^ (z >> 16);
}

HFSM2_CONSTEXPR(14)
BaseRandomT<8>::BaseRandomT(SimpleRandom&& simple) noexcept
	: _state{simple.uint64(), simple.uint64(), simple.uint64(), simple.uint64()}
{}

HFSM2_CONSTEXPR(14)
void
BaseRandomT<8>::seed(SimpleRandom&& simple) noexcept {
_state[0] = simple.uint64();
_state[1] = simple.uint64();
_state[2] = simple.uint64();
_state[3] = simple.uint64();
}

HFSM2_CONSTEXPR(14)
BaseRandomT<8>::BaseRandomT() noexcept
	: BaseRandomT{SimpleRandom{0}}
{}

HFSM2_CONSTEXPR(14)
BaseRandomT<8>::BaseRandomT(const uint64_t s) noexcept
	: BaseRandomT{SimpleRandom{s}}
{}

HFSM2_CONSTEXPR(14)
BaseRandomT<8>::BaseRandomT(const uint64_t(& s)[4]) noexcept
: _state{s[0], s[1], s[2], s[3]}
{}

HFSM2_CONSTEXPR(14)
void
BaseRandomT<8>::seed(const uint64_t s) noexcept {
seed(SimpleRandom{s});
}

HFSM2_CONSTEXPR(14)
void
BaseRandomT<8>::seed(const uint64_t(& s)[4]) noexcept {
_state[0] = s[0];
_state[1] = s[1];
_state[2] = s[2];
_state[3] = s[3];
}

HFSM2_CONSTEXPR(14)
BaseRandomT<4>::BaseRandomT(SimpleRandom&& simple) noexcept
	: _state{simple.uint32(), simple.uint32(), simple.uint32(), simple.uint32()}
{}

HFSM2_CONSTEXPR(14)
void
BaseRandomT<4>::seed(SimpleRandom&& simple) noexcept {
_state[0] = simple.uint32();
_state[1] = simple.uint32();
_state[2] = simple.uint32();
_state[3] = simple.uint32();
}

HFSM2_CONSTEXPR(14)
BaseRandomT<4>::BaseRandomT() noexcept
	: BaseRandomT{SimpleRandom{0}}
{}

HFSM2_CONSTEXPR(14)
BaseRandomT<4>::BaseRandomT(const uint32_t s) noexcept
	: BaseRandomT{SimpleRandom{s}}
{}

HFSM2_CONSTEXPR(14)
BaseRandomT<4>::BaseRandomT(const uint32_t(& s)[4]) noexcept
: _state{s[0], s[1], s[2], s[3]}
{}

HFSM2_CONSTEXPR(14)
void
BaseRandomT<4>::seed(const uint32_t s) noexcept {
seed(SimpleRandom{s});
}

HFSM2_CONSTEXPR(14)
void
BaseRandomT<4>::seed(const uint32_t(& s)[4]) noexcept {
_state[0] = s[0];
_state[1] = s[1];
_state[2] = s[2];
_state[3] = s[3];
}

HFSM2_CONSTEXPR(14)
uint64_t
FloatRandomT<8>::uint64() noexcept {
const uint64_t result = _state[0] + _state[3];

const uint64_t t = _state[1] << 17;

_state[2] ^= _state[0];
_state[3] ^= _state[1];
_state[1] ^= _state[2];
_state[0] ^= _state[3];

_state[2] ^= t;

_state[3] = rotl(_state[3], 45);

return result;
}

HFSM2_CONSTEXPR(14)
void
FloatRandomT<8>::jump() noexcept {
constexpr uint64_t JUMP[] = {
	0x180ec6d33cfd0aba,
	0xd5a61266f0c9392c,
	0xa9582618e03fc9aa,
	0x39abdc4529b1661c
};

uint64_t s0 = 0;
uint64_t s1 = 0;
uint64_t s2 = 0;
uint64_t s3 = 0;

for (unsigned i = 0; i < count<unsigned>(JUMP); ++i)
for (int b = 0; b < 64; ++b) {
if (JUMP[i] & UINT64_C(1) << b) {
s0 ^= _state[0];
s1 ^= _state[1];
s2 ^= _state[2];
s3 ^= _state[3];
			}
			uint64();
		}

_state[0] = s0;
_state[1] = s1;
_state[2] = s2;
_state[3] = s3;
}

HFSM2_CONSTEXPR(14)
uint32_t
FloatRandomT<4>::uint32() noexcept {
const uint32_t result = _state[0] + _state[3];

const uint32_t t = _state[1] << 9;

_state[2] ^= _state[0];
_state[3] ^= _state[1];
_state[1] ^= _state[2];
_state[0] ^= _state[3];

_state[2] ^= t;

_state[3] = rotl(_state[3], 11);

return result;
}

HFSM2_CONSTEXPR(14)
void
FloatRandomT<4>::jump() noexcept {
constexpr uint32_t JUMP[] = {
	0x8764000b,
	0xf542d2d3,
	0x6fa035c3,
	0x77f2db5b
};

uint32_t s0 = 0;
uint32_t s1 = 0;
uint32_t s2 = 0;
uint32_t s3 = 0;

for (unsigned i = 0; i < count<unsigned>(JUMP); ++i)
for (unsigned b = 0; b < 32; ++b) {
if (JUMP[i] & UINT32_C(1) << b) {
s0 ^= _state[0];
s1 ^= _state[1];
s2 ^= _state[2];
s3 ^= _state[3];
			}
			uint32();
		}

_state[0] = s0;
_state[1] = s1;
_state[2] = s2;
_state[3] = s3;
}

HFSM2_CONSTEXPR(14)
uint64_t
IntRandomT<8>::uint64() noexcept {
const uint64_t result = rotl(_state[1] * 5, 7) * 9;

const uint64_t t = _state[1] << 17;

_state[2] ^= _state[0];
_state[3] ^= _state[1];
_state[1] ^= _state[2];
_state[0] ^= _state[3];

_state[2] ^= t;

_state[3] = rotl(_state[3], 45);

return result;
}

HFSM2_CONSTEXPR(14)
void
IntRandomT<8>::jump() noexcept {
constexpr uint64_t JUMP[] = {
	0x180ec6d33cfd0aba,
	0xd5a61266f0c9392c,
	0xa9582618e03fc9aa,
	0x39abdc4529b1661c
};

uint64_t s0 = 0;
uint64_t s1 = 0;
uint64_t s2 = 0;
uint64_t s3 = 0;

for (unsigned i = 0; i < count<unsigned>(JUMP); ++i)
for (int b = 0; b < 64; ++b) {
if (JUMP[i] & UINT64_C(1) << b) {
s0 ^= _state[0];
s1 ^= _state[1];
s2 ^= _state[2];
s3 ^= _state[3];
			}
			uint64();
		}

_state[0] = s0;
_state[1] = s1;
_state[2] = s2;
_state[3] = s3;
}

HFSM2_CONSTEXPR(14)
uint32_t
IntRandomT<4>::uint32() noexcept {
const uint32_t result = rotl(_state[1] * 5, 7) * 9;

const uint32_t t = _state[1] << 9;

_state[2] ^= _state[0];
_state[3] ^= _state[1];
_state[1] ^= _state[2];
_state[0] ^= _state[3];

_state[2] ^= t;

_state[3] = rotl(_state[3], 11);

return result;
}

HFSM2_CONSTEXPR(14)
void
IntRandomT<4>::jump() noexcept {
constexpr uint32_t JUMP[] = {
	0x8764000b,
	0xf542d2d3,
	0x6fa035c3,
	0x77f2db5b
};

uint32_t s0 = 0;
uint32_t s1 = 0;
uint32_t s2 = 0;
uint32_t s3 = 0;

for (unsigned i = 0; i < count<unsigned>(JUMP); ++i)
for (unsigned b = 0; b < 32; ++b) {
if (JUMP[i] & UINT32_C(1) << b) {
s0 ^= _state[0];
s1 ^= _state[1];
s2 ^= _state[2];
s3 ^= _state[3];
			}
			uint32();
		}

_state[0] = s0;
_state[1] = s1;
_state[2] = s2;
_state[3] = s3;
}

}
}

#endif

namespace hfsm2 {
	namespace detail {

		template <typename... Ts>
		struct TL_ final {
		static constexpr Long SIZE = sizeof...(Ts);
	};

	template <Long N>
	struct Const {
		static constexpr Long VALUE = N;
	};

	template <typename, typename>
	struct PrependT;

	template <typename T, typename... Ts>
	struct PrependT<T, TL_<Ts...>> final {
		using Type = TL_<T, Ts...>;
	};

	template <typename... Ts>
	using PrependTypes = typename PrependT<Ts...>::Type;

	template <typename, typename>
	struct MergeT;

	template <typename... Ts1, typename... Ts2>
	struct MergeT<TL_<Ts1...>, TL_<Ts2...>> final {
		using Type = TL_<Ts1..., Ts2...>;
	};

	template <typename... Ts>
	using Merge = typename MergeT<Ts...>::Type;

	template <Long, Long, typename...>
	struct LowerT;

	template <Long NHalf, Long NIndex, typename... Ts>
	using LowerTypes = typename LowerT<NHalf, NIndex, Ts...>::Type;

	template <Long NHalf, Long NIndex, typename TFirst, typename... TRest>
	struct LowerT<NHalf, NIndex, TFirst, TRest...> final {
		using LTypeList = typename LowerT<NHalf, NIndex + 1, TRest...>::Type;

		using Type = Conditional<
			(NIndex < NHalf),
			PrependTypes<TFirst, LTypeList>,
			LTypeList
			>;
	};

	template <Long NHalf, Long NIndex>
	struct LowerT<NHalf, NIndex> final {
		using Type = TL_<>;
	};

	template <typename... Ts>
	using LHalfTypes = LowerTypes<sizeof...(Ts) / 2, 0, Ts...>;

	template <Long, Long, typename...>
	struct UpperT;

	template <Long NHalf, Long NIndex, typename... Ts>
	using UpperTypes = typename UpperT<NHalf, NIndex, Ts...>::Type;

	template <Long NHalf, Long NIndex, typename TFirst, typename... TRest>
	struct UpperT<NHalf, NIndex, TFirst, TRest...> final {
		using Type = Conditional<
			(NIndex < NHalf),
			UpperTypes<NHalf, NIndex + 1, TRest...>,
		TL_<TFirst, TRest...>
		>;
	};

	template <Long NHalf, Long NIndex>
	struct UpperT<NHalf, NIndex> final {
		using Type = TL_<>;
	};

	template <typename... Ts>
	using RHalfTypes = UpperTypes<sizeof...(Ts) / 2, 0, Ts...>;

	template<Long, typename...>
	struct FindImpl
		: Const<INVALID_LONG>
	{};

	template<Long N, typename T, typename TFirst, typename... TRest>
	struct FindImpl<N	 , T, TFirst, TRest...>
		:  FindImpl<N + 1, T,		  TRest...>
	{};

	template<Long N, typename T, typename... Ts>
	struct FindImpl<N, T, T, Ts...>
		: Const<N>
	{};

	template <typename, typename>
	struct Find;

	template <typename T, typename... Ts>
	struct Find<TL_<Ts...>, T> final
		: FindImpl<0, T, Ts...>
	{};

}

template <typename TList, typename T>
constexpr Long index   () noexcept	{ return detail::Find<TList, T>::VALUE;		}

template <typename TList, typename T>
constexpr bool contains() noexcept	{ return index<TList, T>() != INVALID_LONG;	}

}

namespace hfsm2 {
	namespace detail {

		template <typename T>
		HFSM2_CONSTEXPR(11)
		T
		filler()																noexcept	{
	return T{};
}

template <>
HFSM2_CONSTEXPR(11)
Short
filler<Short>()															noexcept	{
return INVALID_SHORT;
}

template <typename T, Long NCapacity>
class StaticArrayT final {
	template <typename>
	friend class IteratorT;

	public:
	using  Iterator	= IteratorT<      StaticArrayT>;
	using CIterator	= IteratorT<const StaticArrayT>;

	using Item		= T;
	using Index		= UCapacity<NCapacity>;

	static constexpr Index CAPACITY	= NCapacity;

	public:
	HFSM2_CONSTEXPR(14)	StaticArrayT() = default;
HFSM2_CONSTEXPR(14)	StaticArrayT(const Item filler)					noexcept	{ fill(filler);						}

	template <typename N>
	HFSM2_CONSTEXPR(14)		  Item& operator[] (const N index)			noexcept;

	template <typename N>
	HFSM2_CONSTEXPR(14)	const Item& operator[] (const N index)	  const noexcept;

	HFSM2_CONSTEXPR(11)	Index count()							  const noexcept	{ return CAPACITY;					}

	HFSM2_CONSTEXPR(14)	void fill(const Item filler)					noexcept;
	HFSM2_CONSTEXPR(14)	void clear()									noexcept	{ fill(filler<Item>());				}
	HFSM2_CONSTEXPR(14)	bool empty()							  const noexcept;

	HFSM2_CONSTEXPR(14)	 Iterator  begin()								noexcept	{ return  Iterator(*this, first());	}
	HFSM2_CONSTEXPR(11)	CIterator  begin()						  const noexcept	{ return CIterator(*this, first());	}
	HFSM2_CONSTEXPR(11)	CIterator cbegin()						  const noexcept	{ return CIterator(*this, first());	}

	HFSM2_CONSTEXPR(14)	 Iterator	 end()								noexcept	{ return  Iterator(*this, limit());	}
	HFSM2_CONSTEXPR(11)	CIterator	 end()						  const noexcept	{ return CIterator(*this, limit());	}
	HFSM2_CONSTEXPR(11)	CIterator	cend()						  const noexcept	{ return CIterator(*this, limit());	}

private:
	HFSM2_CONSTEXPR(11)	Index first()							  const noexcept	{ return 0;							}
	HFSM2_CONSTEXPR(11)	Index  next(const Index index)			  const noexcept	{ return index + 1;					}
	HFSM2_CONSTEXPR(11)	Index limit()							  const noexcept	{ return CAPACITY;					}

private:
Item _items[CAPACITY] {};
};

template <typename T>
struct StaticArrayT<T, 0> final {
	using Item		= T;

	HFSM2_CONSTEXPR(11)	StaticArrayT() = default;
HFSM2_CONSTEXPR(11)	StaticArrayT(const Item)						noexcept	{}
};

template <typename T, Long NCapacity>
class DynamicArrayT final {
	template <typename>
	friend class IteratorT;

	public:
	using  Iterator	= IteratorT<      DynamicArrayT>;
	using CIterator	= IteratorT<const DynamicArrayT>;

	using Item		= T;
	using Index		= UCapacity<NCapacity>;

	static constexpr Index CAPACITY	= NCapacity;

	public:
	template <typename... TArgs>
	HFSM2_CONSTEXPR(14)	Index emplace(const TArgs &... args)				noexcept;

	template <typename... TArgs>
	HFSM2_CONSTEXPR(14)	Index emplace(		TArgs&&... args)				noexcept;

	template <typename N>
	HFSM2_CONSTEXPR(14)		  Item& operator[] (const N index)				noexcept;

	template <typename N>
	HFSM2_CONSTEXPR(14)	const Item& operator[] (const N index)		  const noexcept;

	HFSM2_CONSTEXPR(11)	Index count()								  const noexcept	{ return _count;					}

HFSM2_CONSTEXPR(14)	 void clear()										noexcept	{ _count = 0;						}
	HFSM2_CONSTEXPR(11)	 bool empty()								  const noexcept	{ return _count == 0;				}

	template <Long N>
	HFSM2_CONSTEXPR(14)	DynamicArrayT& operator += (const DynamicArrayT<Item, N>& other)	noexcept;

	HFSM2_CONSTEXPR(14)	 Iterator  begin()									noexcept	{ return  Iterator(*this, first());	}
	HFSM2_CONSTEXPR(11)	CIterator  begin()							  const noexcept	{ return CIterator(*this, first());	}
	HFSM2_CONSTEXPR(11)	CIterator cbegin()							  const noexcept	{ return CIterator(*this, first());	}

	HFSM2_CONSTEXPR(14)	 Iterator	 end()									noexcept	{ return  Iterator(*this, limit());	}
	HFSM2_CONSTEXPR(11)	CIterator	 end()							  const noexcept	{ return CIterator(*this, limit());	}
	HFSM2_CONSTEXPR(11)	CIterator	cend()							  const noexcept	{ return CIterator(*this, limit());	}

private:
	HFSM2_CONSTEXPR(11)	Index first()								  const noexcept	{ return 0;							}
	HFSM2_CONSTEXPR(11)	Index next(const Index index)				  const noexcept	{ return index + 1;					}
	HFSM2_CONSTEXPR(11)	Index limit()								  const noexcept	{ return _count;					}

private:
Index _count = 0;

#ifdef _MSC_VER
#pragma warning(push)
#pragma warning(disable: 4324) // structure was padded due to alignment specifier
#endif

Item _items[CAPACITY] {};

#ifdef _MSC_VER
#pragma warning(pop)
#endif
};

template <typename T>
class DynamicArrayT<T, 0> final {
	public:
	using Item	= T;
	using Index	= UCapacity<0>;

	static constexpr Index CAPACITY = 0;
};

}
}

namespace hfsm2 {
	namespace detail {

		template <typename T, Long NC_>
		template <typename N>
		HFSM2_CONSTEXPR(14)
		T&
		StaticArrayT<T, NC_>::operator[] (const N index) noexcept {
		HFSM2_ASSERT(0 <= index && index < CAPACITY);

		return _items[static_cast<Index>(index)];
	}

	template <typename T, Long NC_>
	template <typename N>
	HFSM2_CONSTEXPR(14)
	const T&
	StaticArrayT<T, NC_>::operator[] (const N index) const noexcept	{
	HFSM2_ASSERT(0 <= index && index < CAPACITY);

	return _items[static_cast<Index>(index)];
}

template <typename T, Long NC_>
HFSM2_CONSTEXPR(14)
void
StaticArrayT<T, NC_>::fill(const Item filler) noexcept {
for (Item& item : _items)
item = filler;
}

template <typename T, Long NC_>
HFSM2_CONSTEXPR(14)
bool
StaticArrayT<T, NC_>::empty() const noexcept {
	for (const Item& item : _items)
		if (item != filler<Item>())
			return false;

	return true;
}

template <typename T, Long NC_>
template <typename... TArgs>
HFSM2_CONSTEXPR(14)
typename DynamicArrayT<T, NC_>::Index
DynamicArrayT<T, NC_>::emplace(const TArgs&... args) noexcept {
	HFSM2_ASSERT(_count < CAPACITY);

new (&_items[_count]) Item{args...};

	return _count++;
}

template <typename T, Long NC_>
template <typename... TArgs>
HFSM2_CONSTEXPR(14)
typename DynamicArrayT<T, NC_>::Index
DynamicArrayT<T, NC_>::emplace(TArgs&&... args) noexcept {
	HFSM2_ASSERT(_count < CAPACITY);

new (&_items[_count]) Item{::hfsm2::forward<TArgs>(args)...};

	return _count++;
}

template <typename T, Long NC_>
template <typename N>
HFSM2_CONSTEXPR(14)
typename DynamicArrayT<T, NC_>::Item&
DynamicArrayT<T, NC_>::operator[] (const N index) noexcept {
	HFSM2_ASSERT(0 <= index && index < _count);

return _items[static_cast<Index>(index)];
}

template <typename T, Long NC_>
template <typename N>
HFSM2_CONSTEXPR(14)
const typename DynamicArrayT<T, NC_>::Item&
DynamicArrayT<T, NC_>::operator[] (const N index) const noexcept {
	HFSM2_ASSERT(0 <= index && index < _count);

return _items[static_cast<Index>(index)];
}

template <typename T, Long NC_>
template <Long N>
HFSM2_CONSTEXPR(14)
DynamicArrayT<T, NC_>&
DynamicArrayT<T, NC_>::operator += (const DynamicArrayT<T, N>& other) noexcept {
	for (const auto& item : other)
		emplace(item);

	return *this;
}

}
}

namespace hfsm2 {
	namespace detail {

		struct Units final {
		HFSM2_CONSTEXPR(11)	Units(Short unit_  = INVALID_SHORT,
		Short width_ = INVALID_SHORT)				noexcept
	: unit {unit_ }
, width{width_}
	{}

Short unit;
Short width;
};

template <unsigned NCapacity>
class BitArrayT final {
	public:
	using Index		= UCapacity<NCapacity>;

	static constexpr Index CAPACITY   = NCapacity;
	static constexpr Index UNIT_COUNT = contain(CAPACITY, 8);

	using BitArray	= BitArrayT<CAPACITY>;

	class Bits {
		template <unsigned>
		friend class BitArrayT;

		private:
		HFSM2_CONSTEXPR(11)	explicit Bits(uint8_t* const storage,
		const Index width)			noexcept
	: _storage{storage}
, _width{width}
		{}

	public:
		HFSM2_CONSTEXPR(14)	explicit operator bool()			  const noexcept;

		HFSM2_CONSTEXPR(14)	void clear()								noexcept;

		template <Short NIndex>
		HFSM2_CONSTEXPR(14)	bool get()							  const noexcept;

		template <Short NIndex>
		HFSM2_CONSTEXPR(14)	void set()									noexcept;

		template <Short NIndex>
		HFSM2_CONSTEXPR(14)	void clear()								noexcept;

		HFSM2_CONSTEXPR(14)	bool get  (const Index index)		  const noexcept;
		HFSM2_CONSTEXPR(14)	void set  (const Index index)				noexcept;
		HFSM2_CONSTEXPR(14)	void clear(const Index index)				noexcept;

	private:
uint8_t* const _storage;
const Index _width;
	};

class CBits {
	template <unsigned>
	friend class BitArrayT;

	private:
	HFSM2_CONSTEXPR(11)	explicit CBits(const uint8_t* const storage,
	const Index width)			noexcept
: _storage{storage}
			, _width{width}
		{}

	public:
		HFSM2_CONSTEXPR(14)	explicit operator bool()			  const noexcept;

		template <Short NIndex>
		HFSM2_CONSTEXPR(14)	bool get()							  const noexcept;

		HFSM2_CONSTEXPR(14)	bool get(const Index index)			  const noexcept;

	private:
const uint8_t* const _storage;
const Index _width;
	};

public:
	HFSM2_CONSTEXPR(14)	BitArrayT()										noexcept	{ clear();	}

	HFSM2_CONSTEXPR(14)	void set()										noexcept;

	HFSM2_CONSTEXPR(14)	void clear()									noexcept;

	template <Short NIndex>
	HFSM2_CONSTEXPR(14)	bool get()								  const noexcept;

	template <Short NIndex>
	HFSM2_CONSTEXPR(14)	void set()										noexcept;

	template <Short NIndex>
	HFSM2_CONSTEXPR(14)	void clear()									noexcept;

	HFSM2_CONSTEXPR(14)	bool empty()							  const noexcept;

	template <typename TIndex>
	HFSM2_CONSTEXPR(14)	bool get  (const TIndex index)			  const noexcept;

	template <typename TIndex>
	HFSM2_CONSTEXPR(14)	void set  (const TIndex index)					noexcept;

	template <typename TIndex>
	HFSM2_CONSTEXPR(14)	void clear(const TIndex index)					noexcept;

	HFSM2_CONSTEXPR(14)	bool operator &  (const BitArray& other)  const noexcept;

	HFSM2_CONSTEXPR(14)	void operator &= (const BitArray& other)		noexcept;

	template <Short NUnit, Short NWidth>
	HFSM2_CONSTEXPR(14)	 Bits  bits()									noexcept;

	template <Short NUnit, Short NWidth>
	HFSM2_CONSTEXPR(14)	CBits cbits()							  const noexcept;

	HFSM2_CONSTEXPR(14)	 Bits  bits(const Units& units)					noexcept;
	HFSM2_CONSTEXPR(14)	CBits cbits(const Units& units)			  const noexcept;

private:
uint8_t _storage[UNIT_COUNT] {};
};

template <>
class BitArrayT<0> final {
	public:
HFSM2_CONSTEXPR(14)	void clear()									noexcept	{}

	HFSM2_CONSTEXPR(11)	bool empty()							  const noexcept	{ return true;	}
};

}
}

namespace hfsm2 {
	namespace detail {

		template <unsigned NCapacity>
		HFSM2_CONSTEXPR(14)
		BitArrayT<NCapacity>::Bits::operator bool() const noexcept {
		const Short fullUnits = _width / 8;

		// TODO: cover this case
		for (Index i = 0; i < fullUnits; ++i)
		if (_storage[i])
		return true;

		const Short bit = _width % 8;
		const uint8_t mask = (1 << bit) - 1;
		const uint8_t& unit = _storage[fullUnits];

		return (unit & mask) != 0;
	}

	template <unsigned NCapacity>
	HFSM2_CONSTEXPR(14)
	void
	BitArrayT<NCapacity>::Bits::clear() noexcept {
	const Index unitCount = contain(_width, 8);

	for (Index i = 0; i < unitCount; ++i)
	_storage[i] = uint8_t{0};
}

template <unsigned NCapacity>
template <Short NIndex>
HFSM2_CONSTEXPR(14)
bool
BitArrayT<NCapacity>::Bits::get() const noexcept {
	constexpr Index INDEX = NIndex;
	HFSM2_ASSERT(INDEX < _width);

	constexpr Index unitIndex = INDEX / 8;
	constexpr Index bitIndex  = INDEX % 8;
	constexpr uint8_t mask = 1 << bitIndex;

	return (_storage[unitIndex] & mask) != 0;
}

template <unsigned NCapacity>
template <Short NIndex>
HFSM2_CONSTEXPR(14)
void
BitArrayT<NCapacity>::Bits::set() noexcept {
constexpr Index INDEX = NIndex;
	HFSM2_ASSERT(INDEX < _width);

constexpr Index unitIndex = INDEX / 8;
constexpr Index bitIndex  = INDEX % 8;
constexpr uint8_t mask = 1 << bitIndex;

_storage[unitIndex] |= mask;
}

template <unsigned NCapacity>
template <Short NIndex>
HFSM2_CONSTEXPR(14)
void
BitArrayT<NCapacity>::Bits::clear() noexcept {
constexpr Index INDEX = NIndex;
	HFSM2_ASSERT(INDEX < _width);

constexpr Index unitIndex = INDEX / 8;
constexpr Index bitIndex  = INDEX % 8;
constexpr uint8_t mask = 1 << bitIndex;

_storage[unitIndex] &= ~mask;
}

template <unsigned NCapacity>
HFSM2_CONSTEXPR(14)
bool
BitArrayT<NCapacity>::Bits::get(const Index index) const noexcept {
	HFSM2_ASSERT(index < _width);

	const Index unit = index / 8;
	const Index bit  = index % 8;
	const uint8_t mask = 1 << bit;

	return (_storage[unit] & mask) != 0;
}

template <unsigned NCapacity>
HFSM2_CONSTEXPR(14)
void
BitArrayT<NCapacity>::Bits::set(const Index index) noexcept {
	HFSM2_ASSERT(index < _width);

const Index unit = index / 8;
const Index bit  = index % 8;
const uint8_t mask = 1 << bit;

_storage[unit] |= mask;
}

template <unsigned NCapacity>
HFSM2_CONSTEXPR(14)
void
BitArrayT<NCapacity>::Bits::clear(const Index index) noexcept {
	HFSM2_ASSERT(index < _width);

const Index unit = index / 8;
const Index bit  = index % 8;
const uint8_t mask = 1 << bit;

_storage[unit] &= ~mask;
}

template <unsigned NCapacity>
HFSM2_CONSTEXPR(14)
BitArrayT<NCapacity>::CBits::operator bool() const noexcept {
const Short fullUnits = _width / 8;

for (Index i = 0; i < fullUnits; ++i)
if (_storage[i])
			return true;

const Short bit = _width % 8;
const uint8_t mask = (1 << bit) - 1;
const uint8_t& unit = _storage[fullUnits];

return (unit & mask) != 0;
}

template <unsigned NCapacity>
template <Short NIndex>
HFSM2_CONSTEXPR(14)
bool
BitArrayT<NCapacity>::CBits::get() const noexcept {
	constexpr Index INDEX = NIndex;
	static_assert(INDEX < _width, "");

	constexpr Index unitIndex = INDEX / 8;
	constexpr Index bitIndex  = INDEX % 8;
	constexpr uint8_t mask = 1 << bitIndex;

	return (_storage[unitIndex] & mask) != 0;
}

template <unsigned NCapacity>
HFSM2_CONSTEXPR(14)
bool
BitArrayT<NCapacity>::CBits::get(const Index index) const noexcept {
	HFSM2_ASSERT(index < _width);

	const Index unit = index / 8;
	const Index bit  = index % 8;
	const uint8_t mask = 1 << bit;

	return (_storage[unit] & mask) != 0;
}

template <unsigned NCapacity>
HFSM2_CONSTEXPR(14)
void
BitArrayT<NCapacity>::set() noexcept {
for (uint8_t& unit : _storage)
unit = UINT8_MAX;
}

template <unsigned NCapacity>
HFSM2_CONSTEXPR(14)
void
BitArrayT<NCapacity>::clear() noexcept {
for (uint8_t& unit : _storage)
unit = uint8_t{0};
}

template <unsigned NCapacity>
HFSM2_CONSTEXPR(14)
bool
BitArrayT<NCapacity>::empty() const noexcept {
	for (const uint8_t& unit : _storage)
		if (unit != uint8_t{0})
		return false;

	return true;
}

template <unsigned NCapacity>
template <Short NIndex>
HFSM2_CONSTEXPR(14)
bool
BitArrayT<NCapacity>::get() const noexcept {
	constexpr Index INDEX = NIndex;
	static_assert(INDEX < CAPACITY, "");

	constexpr Index unitIndex = INDEX / 8;
	constexpr Index bitIndex  = INDEX % 8;
	constexpr uint8_t mask = 1 << bitIndex;

	return (_storage[unitIndex] & mask) != 0;
}

template <unsigned NCapacity>
template <Short NIndex>
HFSM2_CONSTEXPR(14)
void
BitArrayT<NCapacity>::set() noexcept {
constexpr Index INDEX = NIndex;
	static_assert(INDEX < CAPACITY, "");

constexpr Index unitIndex = INDEX / 8;
constexpr Index bitIndex  = INDEX % 8;
constexpr uint8_t mask = 1 << bitIndex;

_storage[unitIndex] |= mask;
}

template <unsigned NCapacity>
template <Short NIndex>
HFSM2_CONSTEXPR(14)
void
BitArrayT<NCapacity>::clear() noexcept {
constexpr Index INDEX = NIndex;
	static_assert(INDEX < CAPACITY, "");

constexpr Index unitIndex = INDEX / 8;
constexpr Index bitIndex  = INDEX % 8;
constexpr uint8_t mask = 1 << bitIndex;

_storage[unitIndex] &= ~mask;
}

template <unsigned NCapacity>
template <typename TIndex>
HFSM2_CONSTEXPR(14)
bool
BitArrayT<NCapacity>::get(const TIndex index) const noexcept {
	HFSM2_ASSERT(index < CAPACITY);

	const Index unit = static_cast<Index>(index) / 8;
	const Index bit  = static_cast<Index>(index) % 8;
	const uint8_t mask = 1 << bit;

	return (_storage[unit] & mask) != 0;
}

template <unsigned NCapacity>
template <typename TIndex>
HFSM2_CONSTEXPR(14)
void
BitArrayT<NCapacity>::set(const TIndex index) noexcept {
	HFSM2_ASSERT(index < CAPACITY);

const Index unit = static_cast<Index>(index) / 8;
const Index bit  = static_cast<Index>(index) % 8;
const uint8_t mask = 1 << bit;

_storage[unit] |= mask;
}

template <unsigned NCapacity>
template <typename TIndex>
HFSM2_CONSTEXPR(14)
void
BitArrayT<NCapacity>::clear(const TIndex index) noexcept {
	HFSM2_ASSERT(index < CAPACITY);

const Index unit = static_cast<Index>(index) / 8;
const Index bit  = static_cast<Index>(index) % 8;
const uint8_t mask = 1 << bit;

_storage[unit] &= ~mask;
}

template <unsigned NCapacity>
HFSM2_CONSTEXPR(14)
bool
BitArrayT<NCapacity>::operator & (const BitArray& other) const noexcept {
for (Index i = 0; i < UNIT_COUNT; ++i)
if ((_storage[i] & other._storage[i]) == 0)
			return false;

	return true;
}

template <unsigned NCapacity>
HFSM2_CONSTEXPR(14)
void
BitArrayT<NCapacity>::operator &= (const BitArray& other) noexcept {
for (Index i = 0; i < UNIT_COUNT; ++i)
_storage[i] &= other._storage[i];
}

template <unsigned NCapacity>
template <Short NUnit, Short NWidth>
HFSM2_CONSTEXPR(14)
typename BitArrayT<NCapacity>::Bits
BitArrayT<NCapacity>::bits() noexcept {
constexpr Short UNIT  = NUnit;
constexpr Short WIDTH = NWidth;
	static_assert(UNIT + contain(WIDTH, 8) <= UNIT_COUNT, "");

return Bits{_storage + UNIT, WIDTH};
}

template <unsigned NCapacity>
template <Short NUnit, Short NWidth>
HFSM2_CONSTEXPR(14)
typename BitArrayT<NCapacity>::CBits
BitArrayT<NCapacity>::cbits() const noexcept {
	constexpr Short UNIT  = NUnit;
	constexpr Short WIDTH = NWidth;
	static_assert(UNIT + contain(WIDTH, 8) <= UNIT_COUNT, "");

	return CBits{_storage + UNIT, WIDTH};
}

template <unsigned NCapacity>
HFSM2_CONSTEXPR(14)
typename BitArrayT<NCapacity>::Bits
BitArrayT<NCapacity>::bits(const Units& units) noexcept {
	HFSM2_ASSERT(units.unit + contain(units.width, 8) <= UNIT_COUNT);

return Bits{_storage + units.unit, units.width};
}

template <unsigned NCapacity>
HFSM2_CONSTEXPR(14)
typename BitArrayT<NCapacity>::CBits
BitArrayT<NCapacity>::cbits(const Units& units) const noexcept {
	HFSM2_ASSERT(units.unit + contain(units.width, 8) <= UNIT_COUNT);

	return CBits{_storage + units.unit, units.width};
}

}
}

namespace hfsm2 {

	enum class Method : uint8_t {
		NONE,

		SELECT,

		//#if HFSM2_UTILITY_THEORY_AVAILABLE()
		RANK,
		UTILITY,
		//#endif

		ENTRY_GUARD,
		ENTER,
		REENTER,
		PRE_UPDATE,
		UPDATE,
		POST_UPDATE,
		PRE_REACT,
		REACT,
		QUERY,
		POST_REACT,
		EXIT_GUARD,
		EXIT,

		//#if HFSM2_PLANS_AVAILABLE()
		PLAN_SUCCEEDED,
		PLAN_FAILED,
		//#endif

		COUNT
	};

	enum class TransitionType : uint8_t {
		CHANGE,
		RESTART,
		RESUME,
		SELECT,

		//#if HFSM2_UTILITY_THEORY_AVAILABLE()
		UTILIZE,
		RANDOMIZE,
		//#endif

		SCHEDULE,

		COUNT
	};

#if HFSM2_PLANS_AVAILABLE()

	enum class StatusEvent : uint8_t {
		SUCCEEDED,
		FAILED,

		COUNT
	};

#endif

	static
	HFSM2_CONSTEXPR(14)
	const char*
	methodName(const Method method)											noexcept	{
	switch (method) {

	case Method::SELECT:		 return "select";

	//#if HFSM2_UTILITY_THEORY_AVAILABLE()
	case Method::RANK:			 return "rank";
	case Method::UTILITY:		 return "utility";
	//#endif

	case Method::ENTRY_GUARD:	 return "entryGuard";
	case Method::ENTER:			 return "enter";
	case Method::REENTER:		 return "reenter";
	case Method::PRE_UPDATE:	 return "preUpdate";
	case Method::UPDATE:		 return "update";
	case Method::POST_UPDATE:	 return "postUpdate";
	case Method::PRE_REACT:		 return "preReact";
	case Method::REACT:			 return "react";
	case Method::POST_REACT:	 return "postReact";
	case Method::QUERY:			 return "query";
	case Method::EXIT_GUARD:	 return "exitGuard";
	case Method::EXIT:			 return "exit";

	//#if HFSM2_PLANS_AVAILABLE()
	case Method::PLAN_SUCCEEDED: return "planSucceeded";
	case Method::PLAN_FAILED:	 return "planFailed";
	//#endif

	default:
	HFSM2_BREAK();
	return nullptr;
}
}

static
HFSM2_CONSTEXPR(14)
const char*
transitionName(const TransitionType type)								noexcept	{
	switch (type) {
	case TransitionType::CHANGE:	return "changeTo";
	case TransitionType::RESTART:	return "restart";
	case TransitionType::RESUME:	return "resume";
	case TransitionType::SELECT:	return "select";

//#if HFSM2_UTILITY_THEORY_AVAILABLE()
	case TransitionType::UTILIZE:	return "utilize";
	case TransitionType::RANDOMIZE:	return "randomize";
//#endif

	case TransitionType::SCHEDULE:	return "schedule";

	default:
		HFSM2_BREAK();
return nullptr;
	}
}

namespace detail {

	enum Strategy {
		Composite,
		Resumable,
		Selectable,

		//#if HFSM2_UTILITY_THEORY_AVAILABLE()
		Utilitarian,
		RandomUtil,
		//#endif
	};

#ifdef _MSC_VER
#pragma warning(push)
#pragma warning(disable: 4324) // structure was padded due to alignment specifier
#endif

	struct TransitionBase {
		HFSM2_CONSTEXPR(11)
		TransitionBase()													noexcept = default;

		HFSM2_CONSTEXPR(11)
		TransitionBase(const StateID destination_,
		const TransitionType type_)							noexcept
	: destination{destination_}
, type		 {type_}
	{}

	HFSM2_CONSTEXPR(11)
	TransitionBase(const StateID origin_,
				   const StateID destination_,
				   const TransitionType type_)							noexcept
		: origin	 {origin_}
		, destination{destination_}
		, type		 {type_}
	{}

	HFSM2_CONSTEXPR(11)
bool
operator == (const TransitionBase& other)					  const noexcept	{
	return origin	   == other.origin		&&
		destination == other.destination &&
		method	   == other.method		&&
		type		   == other.type;
}

	HFSM2_CONSTEXPR(11)
bool
operator != (const TransitionBase& other)					  const noexcept	{
	return origin	   != other.origin		||
		destination != other.destination ||
		method	   != other.method		||
		type		   != other.type;
}

StateID	origin		= INVALID_STATE_ID;
StateID	destination	= INVALID_STATE_ID;
Method	method		= Method::NONE;
TransitionType type	= TransitionType::COUNT;
};

#ifdef _MSC_VER
#pragma warning(pop)
#endif

template <typename TPayload>
struct TransitionT final
	: TransitionBase
	{
	using Payload = TPayload;
	using Storage = uint8_t[sizeof(Payload)];

	using TransitionBase::TransitionBase;

	HFSM2_CONSTEXPR(14)
	TransitionT()														noexcept	{
new (&storage) Payload{};
	}

	HFSM2_CONSTEXPR(14)
	TransitionT(const StateID destination_,
				const TransitionType type_,
				const Payload& payload)									noexcept
: TransitionBase{destination_, type_}
		, payloadSet{true}
	{
		new (&storage) Payload{payload};
	}

	HFSM2_CONSTEXPR(14)
	TransitionT(const StateID origin_,
				const StateID destination_,
				const TransitionType type_,
				const Payload& payload)									noexcept
: TransitionBase{origin_, destination_, type_}
		, payloadSet{true}
	{
		new (&storage) Payload{payload};
	}

	HFSM2_CONSTEXPR(11)
bool
operator == (const TransitionT& other)						  const noexcept	{
	return TransitionBase::operator == (other) &&
		(payloadSet ==  other.payloadSet);
	//	  (!payloadSet && !other.payloadSet || payload ==  other.payload);
}

	HFSM2_CONSTEXPR(11)
bool
operator != (const TransitionT& other)						  const noexcept	{
	return TransitionBase::operator != (other) ||
		(payloadSet != other.payloadSet);
	//	   (payloadSet |= other.payloadSet || payload != other.payload);
}

	HFSM2_CONSTEXPR(11)
const Payload*
payload()													  const noexcept	{
	return payloadSet ?
		reinterpret_cast<const Payload*>(&storage) : nullptr;
}

#ifdef _MSC_VER
#pragma warning(push)
#pragma warning(disable: 4324) // structure was padded due to alignment specifier
#endif

	alignas(Payload) Storage storage {};

#ifdef _MSC_VER
#pragma warning(pop)
#endif

bool payloadSet = false;
};

template <>
struct TransitionT<void> final
	: TransitionBase
{
	using TransitionBase::TransitionBase;
};

}

struct Request final {
TransitionType type;
Short index;
};

}

namespace hfsm2 {

	struct HFSM2_EMPTY_BASES EmptyContext {};

#if HFSM2_LOG_INTERFACE_AVAILABLE()

template <
	FeatureTag NFeatureTag = HFSM2_FEATURE_TAG
  , typename TContext = EmptyContext
HFSM2_IF_UTILITY_THEORY(, typename TUtilty = float)
>
struct LoggerInterfaceT {
	using Context		 = TContext;

#if HFSM2_UTILITY_THEORY_AVAILABLE()
	using Utilty		 = TUtilty;
#endif

	using Method		 = ::hfsm2::Method;
	using Prong			 = ::hfsm2::Prong;
	using StateID		 = ::hfsm2::StateID;
	using TransitionType = ::hfsm2::TransitionType;

#if HFSM2_PLANS_AVAILABLE()
	using StatusEvent	 = ::hfsm2::StatusEvent;
#endif

	HFSM2_CONSTEXPR(NO)
	virtual
	void
	recordMethod(const Context& HFSM2_UNUSED(context),
	const StateID HFSM2_UNUSED(origin),
	const Method HFSM2_UNUSED(method))
{}

	HFSM2_CONSTEXPR(NO)
	virtual
	void
	recordTransition(const Context& HFSM2_UNUSED(context),
					 const StateID HFSM2_UNUSED(origin),
					 const TransitionType HFSM2_UNUSED(transitionType),
					 const StateID HFSM2_UNUSED(target))
	{}

#if HFSM2_PLANS_AVAILABLE()

	HFSM2_CONSTEXPR(NO)
	virtual
	void
	recordTaskStatus(const Context& HFSM2_UNUSED(context),
					 const StateID HFSM2_UNUSED(region),
					 const StateID HFSM2_UNUSED(origin),
					 const StatusEvent HFSM2_UNUSED(event))
	{}

	HFSM2_CONSTEXPR(NO)
	virtual
	void
	recordPlanStatus(const Context& HFSM2_UNUSED(context),
					 const StateID HFSM2_UNUSED(region),
					 const StatusEvent HFSM2_UNUSED(event))
	{}

#endif

	HFSM2_CONSTEXPR(NO)
	virtual
	void
	recordCancelledPending(const Context& HFSM2_UNUSED(context),
						   const StateID HFSM2_UNUSED(origin))
	{}

	HFSM2_CONSTEXPR(NO)
	virtual
	void
	recordSelectResolution(const Context& HFSM2_UNUSED(context),
						   const StateID HFSM2_UNUSED(head),
						   const Prong HFSM2_UNUSED(prong))
	{}

#if HFSM2_UTILITY_THEORY_AVAILABLE()

	HFSM2_CONSTEXPR(NO)
	virtual
	void
	recordUtilityResolution(const Context& HFSM2_UNUSED(context),
							const StateID HFSM2_UNUSED(head),
							const Prong HFSM2_UNUSED(prong),
							const Utilty HFSM2_UNUSED(utilty))
	{}

	HFSM2_CONSTEXPR(NO)
	virtual
	void
	recordRandomResolution(const Context& HFSM2_UNUSED(context),
						   const StateID HFSM2_UNUSED(head),
						   const Prong HFSM2_UNUSED(prong),
						   const Utilty HFSM2_UNUSED(utilty))
	{}

#endif
};

#else

template <
	FeatureTag NFeatureTag = HFSM2_FEATURE_TAG
  , typename TContext = EmptyContext
HFSM2_IF_UTILITY_THEORY(, typename TUtilty = float)
>
using LoggerInterfaceT = void;

#endif

using LoggerInterface = LoggerInterfaceT<>;

}

#if HFSM2_STRUCTURE_REPORT_AVAILABLE()

namespace hfsm2 {

	struct StructureEntry final {
	bool isActive;
	const wchar_t* prefix;
	const char* name;
};

namespace detail {

	enum class RegionType {
		COMPOSITE,
		ORTHOGONAL,

		COUNT
	};

	struct StructureStateInfo final {
	StructureStateInfo() noexcept = default;

	HFSM2_CONSTEXPR(11)
	StructureStateInfo(const Long parent_,
	const RegionType regionType_,
	const Short depth_,
	const char* const name_)							noexcept
: name{name_}
		, parent{parent_}
		, regionType{regionType_ }
		, depth{depth_}
	{}

const char* name	  = nullptr;
Long parent			  = INVALID_LONG;
RegionType regionType = RegionType::COUNT;
Short depth			  = INVALID_SHORT;
};

}
}

#endif

#if HFSM2_PLANS_AVAILABLE()

namespace hfsm2 {
namespace detail {

struct TaskBase {
	static_assert(sizeof(Long) == sizeof(StateID), "");

	HFSM2_CONSTEXPR(11)	TaskBase()										noexcept	{}

	HFSM2_CONSTEXPR(11)	TaskBase(const StateID origin_,
								 const StateID destination_,
								 const TransitionType type_)			noexcept
		: origin{origin_}
		, destination{destination_}
		, type{type_}
	{}

	HFSM2_CONSTEXPR(11) bool cyclic()							  const noexcept	{ return origin == destination;	}

union {
	StateID origin		= INVALID_STATE_ID;
	Long prev;
};

union {
	StateID destination	= INVALID_STATE_ID;
	Long next;
};

TransitionType type = TransitionType::COUNT;
};

HFSM2_CONSTEXPR(11)
bool
	operator == (const TaskBase& lhs,
	const TaskBase& rhs)										noexcept
{
	return lhs.origin	   == rhs.origin &&
		lhs.destination == rhs.destination &&
		lhs.type		   == rhs.type;
}

template <typename TPayload>
struct TaskT final
	: TaskBase
	{
	using Payload = TPayload;
	using Storage = uint8_t[sizeof(Payload)];

	using TaskBase::TaskBase;

	HFSM2_CONSTEXPR(14)	TaskT()											noexcept	{
new (&storage) Payload{};
	}

	HFSM2_CONSTEXPR(14)	TaskT(const StateID origin_,
							  const StateID destination_,
							  const TransitionType type_,
							  const Payload& payload)					noexcept
: TaskBase{origin_, destination_, type_}
		, payloadSet{true}
	{
		new (&storage) Payload{payload};
	}

	HFSM2_CONSTEXPR(11)
const Payload*
payload()													  const noexcept	{
	return payloadSet ?
		reinterpret_cast<const Payload*>(&storage) : nullptr;
}

#ifdef _MSC_VER
#pragma warning(push)
#pragma warning(disable: 4324) // structure was padded due to alignment specifier
#endif

	alignas(Payload) Storage storage {};

#ifdef _MSC_VER
#pragma warning(pop)
#endif

bool payloadSet = false;
};

template <>
struct TaskT<void> final
	: TaskBase
{
	using TaskBase::TaskBase;
};

}
}

#endif

#if HFSM2_PLANS_AVAILABLE()

namespace hfsm2 {
namespace detail {

template <typename TPayload, Long NCapacity>
class TaskListT {
public:
	using Index		= Long;

	static constexpr Index CAPACITY	= NCapacity;
	static constexpr Index INVALID	= Index (-1);

private:
	using Payload	= TPayload;
	using Item		= TaskT<Payload>;

public:
	HFSM2_CONSTEXPR(14)	 void clear()											noexcept;

	template <typename... TArgs>
	HFSM2_CONSTEXPR(14)	Index emplace(TArgs&&... args)							noexcept;

	HFSM2_CONSTEXPR(14)	void remove(const Index i)								noexcept;

	HFSM2_CONSTEXPR(14)		  Item& operator[] (const Index i)					noexcept;
	HFSM2_CONSTEXPR(11)	const Item& operator[] (const Index i)			  const noexcept;

	HFSM2_CONSTEXPR(11)	Index count()									  const noexcept	{ return _count;		}
	HFSM2_CONSTEXPR(11)	bool  empty()									  const noexcept	{ return _count == 0;	}

private:
	HFSM2_IF_ASSERT(void verifyStructure(const Index occupied = INVALID)  const noexcept);

private:
	Index _vacantHead = 0;
	Index _vacantTail = 0;
	Index _last		  = 0;
	Index _count	  = 0;
	Item _items[CAPACITY] {};
};

template <typename TItem>
class TaskListT<TItem, 0> {};

}
}

#if HFSM2_PLANS_AVAILABLE()

namespace hfsm2 {
namespace detail {

template <typename TP_, Long NC_>
HFSM2_CONSTEXPR(14)
void
TaskListT<TP_, NC_>::clear() noexcept {
	_vacantHead	= 0;
	_vacantTail	= 0;
	_last		= 0;
	_count		= 0;
}

template <typename TP_, Long NC_>
template <typename... TA_>
HFSM2_CONSTEXPR(14)
Long
TaskListT<TP_, NC_>::emplace(TA_&&... args) noexcept {
	HFSM2_ASSERT(_last  <= CAPACITY);

	if (_count < CAPACITY) {
		HFSM2_ASSERT(_vacantHead < CAPACITY);
		HFSM2_ASSERT(_vacantTail < CAPACITY);

		const Index index = _vacantHead;
		Item& item = _items[index];

		if (_vacantHead != _vacantTail) {
			// recycle
			HFSM2_ASSERT(item.prev == INVALID);
			HFSM2_ASSERT(item.next != INVALID);

			_vacantHead = item.next;

			Item& head = _items[_vacantHead];
			HFSM2_ASSERT(head.prev == index);
			head.prev = INVALID;
		} else if (_last < CAPACITY - 1) {
			// grow
			++_last;
			_vacantHead = _last;
			_vacantTail = _last;

			Item& vacant = _items[_vacantHead];
			vacant.prev = INVALID;
			vacant.next = INVALID;
		} else {
			// last
			HFSM2_ASSERT(_count == CAPACITY - 1);

			_last = CAPACITY;
_vacantHead = INVALID;
_vacantTail = INVALID;
		}

		new (&item) Item{::hfsm2::forward<TA_>(args)...};
++_count;

		HFSM2_IF_ASSERT(verifyStructure());

return index;
	} else {
		// full
		HFSM2_ASSERT(_vacantHead == INVALID);
		HFSM2_ASSERT(_vacantTail == INVALID);
		HFSM2_ASSERT(_count		 == CAPACITY);
		HFSM2_BREAK();

return INVALID;
	}
}

template <typename TP_, Long NC_>
HFSM2_CONSTEXPR(14)
void
TaskListT<TP_, NC_>::remove(const Index i) noexcept {
	HFSM2_ASSERT(i < CAPACITY && _count);

Item& item = _items[i];

	if (_count < CAPACITY) {
		HFSM2_ASSERT(_vacantHead < CAPACITY);
		HFSM2_ASSERT(_vacantTail < CAPACITY);

item.prev = INVALID;
item.next = _vacantHead;

Item& head = _items[_vacantHead];
head.prev = i;

_vacantHead = i;
	} else {
		// 0 -> 1
		HFSM2_ASSERT(_count		 == CAPACITY);
		HFSM2_ASSERT(_vacantHead == INVALID);
		HFSM2_ASSERT(_vacantTail == INVALID);

item.prev = INVALID;
item.next = INVALID;

_vacantHead = i;
_vacantTail = i;
	}

--_count;

	HFSM2_IF_ASSERT(verifyStructure());
}

template <typename TP_, Long NC_>
HFSM2_CONSTEXPR(14)
typename TaskListT<TP_, NC_>::Item&
TaskListT<TP_, NC_>::operator[] (const Index i) noexcept {
	HFSM2_IF_ASSERT(verifyStructure());

return _items[i];
}

template <typename TP_, Long NC_>
HFSM2_CONSTEXPR(11)
const typename TaskListT<TP_, NC_>::Item&
TaskListT<TP_, NC_>::operator[] (const Index i) const noexcept {
	HFSM2_IF_ASSERT(verifyStructure());

return _items[i];
}

#if HFSM2_ASSERT_AVAILABLE()

template <typename TP_, Long NC_>
void
TaskListT<TP_, NC_>::verifyStructure(const Index occupied) const noexcept {
	if (_count < CAPACITY) {
		HFSM2_ASSERT(_vacantHead < CAPACITY);
		HFSM2_ASSERT(_vacantTail < CAPACITY);

		HFSM2_ASSERT(_items[_vacantHead].prev == INVALID);
		HFSM2_ASSERT(_items[_vacantTail].next == INVALID);

		Index emptyCount = 1;

		for (Index c = _vacantHead; c != _vacantTail; ) {
			HFSM2_ASSERT(occupied != c);

			const Item& current = _items[c];

			const Long f = current.next;
			if (f != INVALID) {
				// next
				const Item& following = _items[f];

				HFSM2_ASSERT(following.prev == c);

				c = f;
				continue;
			} else {
				// end
				HFSM2_ASSERT(_vacantTail == c);
				HFSM2_ASSERT(_count		 == CAPACITY - emptyCount);

				break;
			}
		}
	} else {
		HFSM2_ASSERT(_vacantHead == INVALID);
		HFSM2_ASSERT(_vacantTail == INVALID);
	}
}

#endif

}
}

#endif

#endif

namespace hfsm2 {
	namespace detail {

		struct alignas(2 * sizeof(ForkID)) Parent final {
		HFSM2_CONSTEXPR(11)
		Parent() = default;

		HFSM2_CONSTEXPR(11)
		Parent(const ForkID forkId_)										noexcept
	: forkId{forkId_}
{}

	HFSM2_CONSTEXPR(11)
	Parent(const ForkID forkId_,
		   const Prong prong_)											noexcept
		: forkId{forkId_}
		, prong{prong_}
	{}

	HFSM2_CONSTEXPR(11)
	explicit operator bool()									  const noexcept	{
		return forkId != INVALID_FORK_ID &&
prong  != INVALID_PRONG;
	}

ForkID forkId = INVALID_FORK_ID;
Prong  prong  = INVALID_PRONG;
};

template <typename TRegistry>
struct BackUpT final {
	using CompoForks = typename TRegistry::CompoForks;
	using OrthoForks = typename TRegistry::OrthoForks;

	CompoForks compoRequested;
	OrthoForks orthoRequested;
	CompoForks compoResumable;
};

template <
	typename
  , typename
  , typename
  , Long
  , Long
  , Long
  , typename
  HFSM2_IF_SERIALIZATION(, Long)
  HFSM2_IF_PLANS(, Long)
  , typename
>
struct ArgsT;

template <typename>
struct RegistryT;

template <
	typename TConfig
  , typename TStateList
  , typename TRegionList
  , Long NCompoCount
  , Long NOrthoCount
  , Long NOrthoUnits
  , typename TReactOrder
  HFSM2_IF_SERIALIZATION(, Long NSerialBits)
  HFSM2_IF_PLANS(, Long NTaskCapacity)
  , typename TPayload
>
struct RegistryT<
		   ArgsT<
			   TConfig
			 , TStateList
			 , TRegionList
			 , NCompoCount
			 , NOrthoCount
			 , NOrthoUnits
			 , TReactOrder
			 HFSM2_IF_SERIALIZATION(, NSerialBits)
			 HFSM2_IF_PLANS(, NTaskCapacity)
			 , TPayload
		   >
	   > final
{
	using StateList		= TStateList;
using RegionList	= TRegionList;

static constexpr Long  STATE_COUNT		= StateList::SIZE;
static constexpr Long  REGION_COUNT		= RegionList::SIZE;
static constexpr Short COMPO_COUNT		= NCompoCount;
static constexpr Short ORTHO_COUNT		= NOrthoCount;
static constexpr Short ORTHO_UNITS		= NOrthoUnits;

	using Payload		= TPayload;
using Transition	= TransitionT<Payload>;

using StateParents	= StaticArrayT<Parent,  STATE_COUNT>;

using CompoParents	= StaticArrayT<Parent,  COMPO_COUNT>;
using OrthoParents	= StaticArrayT<Parent,  ORTHO_COUNT>;
using OrthoUnits	= StaticArrayT<Units,   ORTHO_UNITS>;
using RegionHeads	= StaticArrayT<StateID, REGION_COUNT>;
using RegionSizes	= StaticArrayT<Long,    REGION_COUNT>;

using CompoForks	= StaticArrayT<Prong,   COMPO_COUNT>;
using OrthoForks	= BitArrayT	  <ORTHO_UNITS * 8>;
using OrthoBits		= typename OrthoForks::Bits;
	using CompoRemains	= BitArrayT	  <COMPO_COUNT>;

using BackUp		= BackUpT	  <RegistryT>;

#if HFSM2_PLANS_AVAILABLE()
	using CompoStatuses	= BitArrayT	  <COMPO_COUNT>;
#endif

	HFSM2_CONSTEXPR(14)	Prong activeSubState		(const StateID stateId)	  const noexcept;

	HFSM2_CONSTEXPR(11)	bool isActive				()						  const noexcept;
	HFSM2_CONSTEXPR(14)	bool isActive				(const StateID stateId)	  const noexcept;
	HFSM2_CONSTEXPR(14)	bool isResumable			(const StateID stateId)	  const noexcept;

	HFSM2_CONSTEXPR(14)	bool isPendingChange		(const StateID stateId)	  const noexcept;
	HFSM2_CONSTEXPR(14)	bool isPendingEnter			(const StateID stateId)	  const noexcept;
	HFSM2_CONSTEXPR(14)	bool isPendingExit			(const StateID stateId)	  const noexcept;

	HFSM2_CONSTEXPR(14)	const Parent& forkParent	(const ForkID forkId)	  const noexcept;

	HFSM2_CONSTEXPR(14)	OrthoBits requestedOrthoFork(const ForkID forkId)			noexcept;

	HFSM2_CONSTEXPR(14)	bool requestImmediate		(const Transition& request)		noexcept;
	HFSM2_CONSTEXPR(14)	void requestScheduled		(const StateID stateId)			noexcept;

	HFSM2_CONSTEXPR(14)	void clearRequests			()								noexcept;
	HFSM2_CONSTEXPR(14)	void clear					()								noexcept;

	HFSM2_CONSTEXPR(11)	bool empty					()						  const noexcept;

StateParents stateParents;
CompoParents compoParents;
OrthoParents orthoParents;
OrthoUnits	 orthoUnits;

RegionHeads	 regionHeads;
RegionSizes	 regionSizes;

CompoForks compoRequested{INVALID_PRONG};
OrthoForks orthoRequested;
CompoForks compoActive	 {INVALID_PRONG};
CompoForks compoResumable{INVALID_PRONG};

CompoRemains compoRemains;

#if HFSM2_PLANS_AVAILABLE()
CompoStatuses compoStatuses;
#endif
};

template <
	typename TConfig
  , typename TStateList
  , typename TRegionList
  , Long NCompoCount
  , typename TReactOrder
  HFSM2_IF_SERIALIZATION(, Long NSerialBits)
  HFSM2_IF_PLANS(, Long NTaskCapacity)
  , typename TPayload
>
struct RegistryT<
		   ArgsT<
			   TConfig
			 , TStateList
			 , TRegionList
			 , NCompoCount
			 , 0
			 , 0
			 , TReactOrder
			 HFSM2_IF_SERIALIZATION(, NSerialBits)
			 HFSM2_IF_PLANS(, NTaskCapacity)
			 , TPayload
		   >
	   > final
{
	using StateList		= TStateList;
using RegionList	= TRegionList;

static constexpr Long  STATE_COUNT		= StateList::SIZE;
static constexpr Long  REGION_COUNT		= RegionList::SIZE;
static constexpr Short COMPO_COUNT		= NCompoCount;

	using Payload		= TPayload;
using Transition	= TransitionT<Payload>;

using StateParents	= StaticArrayT<Parent,  STATE_COUNT>;
using CompoParents	= StaticArrayT<Parent,  COMPO_COUNT>;
using RegionHeads	= StaticArrayT<StateID, REGION_COUNT>;
using RegionSizes	= StaticArrayT<Long,    REGION_COUNT>;

using CompoForks	= StaticArrayT<Prong,   COMPO_COUNT>;
using OrthoForks	= BitArrayT	  <0>;
using CompoRemains	= BitArrayT	  <COMPO_COUNT>;

using BackUp		= BackUpT	  <RegistryT>;

#if HFSM2_PLANS_AVAILABLE()
	using CompoStatuses	= BitArrayT	  <COMPO_COUNT>;
#endif

	HFSM2_CONSTEXPR(14)	Prong activeSubState	(const StateID stateId)	  const noexcept;

	HFSM2_CONSTEXPR(11)	bool isActive			()						  const noexcept;
	HFSM2_CONSTEXPR(14)	bool isActive			(const StateID stateId)	  const noexcept;
	HFSM2_CONSTEXPR(14)	bool isResumable		(const StateID stateId)	  const noexcept;

	HFSM2_CONSTEXPR(14)	bool isPendingChange	(const StateID stateId)	  const noexcept;
	HFSM2_CONSTEXPR(14)	bool isPendingEnter		(const StateID stateId)	  const noexcept;
	HFSM2_CONSTEXPR(14)	bool isPendingExit		(const StateID stateId)	  const noexcept;

	HFSM2_CONSTEXPR(14)	const Parent& forkParent(const ForkID forkId)	  const noexcept;

	HFSM2_CONSTEXPR(14)	bool requestImmediate	(const Transition& request)		noexcept;
	HFSM2_CONSTEXPR(14)	void requestScheduled	(const StateID stateId)			noexcept;

	HFSM2_CONSTEXPR(14)	void clearRequests		()								noexcept;
	HFSM2_CONSTEXPR(14)	void clear				()								noexcept;

	HFSM2_CONSTEXPR(11)	bool empty				()						  const noexcept;

StateParents stateParents;
CompoParents compoParents;

RegionHeads	 regionHeads;
RegionSizes	 regionSizes;

CompoForks compoRequested{INVALID_PRONG};
OrthoForks orthoRequested;
CompoForks compoActive	 {INVALID_PRONG};
CompoForks compoResumable{INVALID_PRONG};

CompoRemains compoRemains;

#if HFSM2_PLANS_AVAILABLE()
CompoStatuses compoStatuses;
#endif
};

template <typename TRegistry>
HFSM2_CONSTEXPR(14)
void
backup(const TRegistry& registry,
	   BackUpT<TRegistry>& copy) noexcept
{
	overwrite(copy.compoRequested, registry.compoRequested);
	overwrite(copy.orthoRequested, registry.orthoRequested);
	overwrite(copy.compoResumable, registry.compoResumable);
}

template <typename TRegistry>
HFSM2_CONSTEXPR(14)
void
restore(TRegistry& registry,
		const BackUpT<TRegistry>& copy) noexcept
{
	overwrite(registry.compoRequested, copy.compoRequested);
	overwrite(registry.orthoRequested, copy.orthoRequested);
	overwrite(registry.compoResumable, copy.compoResumable);
}

}
}

namespace hfsm2 {
	namespace detail {

		template <typename TG_, typename TSL_, typename TRL_, Long NCC_, Long NOC_, Long NOU_, typename TRO_ HFSM2_IF_SERIALIZATION(, Long NSB_) HFSM2_IF_PLANS(, Long NTC_), typename TTP_>
		HFSM2_CONSTEXPR(14)
		Prong
		RegistryT<ArgsT<TG_, TSL_, TRL_, NCC_, NOC_, NOU_, TRO_ HFSM2_IF_SERIALIZATION(, NSB_) HFSM2_IF_PLANS(, NTC_), TTP_>>::activeSubState(const StateID stateId) const noexcept {
		const StateID subStateId = stateId + 1;

		if (HFSM2_CHECKED(	 stateId < STATE_COUNT) &&
		HFSM2_CHECKED(subStateId < STATE_COUNT))
		{
		if (const Parent parent = stateParents[subStateId]) {
		HFSM2_ASSERT(parent.forkId != 0);

		if (parent.forkId > 0)
		return compoActive[parent.forkId - 1];
	}
}

	return INVALID_PRONG;
}

template <typename TG_, typename TSL_, typename TRL_, Long NCC_, Long NOC_, Long NOU_, typename TRO_ HFSM2_IF_SERIALIZATION(, Long NSB_) HFSM2_IF_PLANS(, Long NTC_), typename TTP_>
HFSM2_CONSTEXPR(11)
bool
RegistryT<ArgsT<TG_, TSL_, TRL_, NCC_, NOC_, NOU_, TRO_ HFSM2_IF_SERIALIZATION(, NSB_) HFSM2_IF_PLANS(, NTC_), TTP_>>::isActive() const noexcept {
return compoActive[ROOT_ID] != INVALID_PRONG;
}

template <typename TG_, typename TSL_, typename TRL_, Long NCC_, Long NOC_, Long NOU_, typename TRO_ HFSM2_IF_SERIALIZATION(, Long NSB_) HFSM2_IF_PLANS(, Long NTC_), typename TTP_>
HFSM2_CONSTEXPR(14)
bool
RegistryT<ArgsT<TG_, TSL_, TRL_, NCC_, NOC_, NOU_, TRO_ HFSM2_IF_SERIALIZATION(, NSB_) HFSM2_IF_PLANS(, NTC_), TTP_>>::isActive(const StateID stateId) const noexcept {
	if (HFSM2_CHECKED(stateId < STATE_COUNT)) {
for (Parent parent = stateParents[stateId];
parent;
parent = forkParent(parent.forkId))
		{
			HFSM2_ASSERT(parent.forkId != 0);

			if (parent.forkId > 0)
return parent.prong == compoActive[parent.forkId - 1];
		}

		return isActive();
	}

	return false;
}

template <typename TG_, typename TSL_, typename TRL_, Long NCC_, Long NOC_, Long NOU_, typename TRO_ HFSM2_IF_SERIALIZATION(, Long NSB_) HFSM2_IF_PLANS(, Long NTC_), typename TTP_>
HFSM2_CONSTEXPR(14)
bool
RegistryT<ArgsT<TG_, TSL_, TRL_, NCC_, NOC_, NOU_, TRO_ HFSM2_IF_SERIALIZATION(, NSB_) HFSM2_IF_PLANS(, NTC_), TTP_>>::isResumable(const StateID stateId) const noexcept {
	if (HFSM2_CHECKED(stateId < STATE_COUNT))
for (Parent parent = stateParents[stateId];
parent;
parent = forkParent(parent.forkId))
		{
			HFSM2_ASSERT(parent.forkId != 0);

			if (parent.forkId > 0)
return parent.prong == compoResumable[parent.forkId - 1];
		}

	return false;
}

template <typename TG_, typename TSL_, typename TRL_, Long NCC_, Long NOC_, Long NOU_, typename TRO_ HFSM2_IF_SERIALIZATION(, Long NSB_) HFSM2_IF_PLANS(, Long NTC_), typename TTP_>
HFSM2_CONSTEXPR(14)
bool
RegistryT<ArgsT<TG_, TSL_, TRL_, NCC_, NOC_, NOU_, TRO_ HFSM2_IF_SERIALIZATION(, NSB_) HFSM2_IF_PLANS(, NTC_), TTP_>>::isPendingChange(const StateID stateId) const noexcept {
	if (HFSM2_CHECKED(stateId < STATE_COUNT))
for (Parent parent = stateParents[stateId];
parent;
parent = forkParent(parent.forkId))
		{
			HFSM2_ASSERT(parent.forkId != 0);

			if (parent.forkId > 0)
return compoRequested[parent.forkId - 1] !=
compoActive	 [parent.forkId - 1];
		}

	return false;
}

template <typename TG_, typename TSL_, typename TRL_, Long NCC_, Long NOC_, Long NOU_, typename TRO_ HFSM2_IF_SERIALIZATION(, Long NSB_) HFSM2_IF_PLANS(, Long NTC_), typename TTP_>
HFSM2_CONSTEXPR(14)
bool
RegistryT<ArgsT<TG_, TSL_, TRL_, NCC_, NOC_, NOU_, TRO_ HFSM2_IF_SERIALIZATION(, NSB_) HFSM2_IF_PLANS(, NTC_), TTP_>>::isPendingEnter(const StateID stateId) const noexcept {
	if (HFSM2_CHECKED(stateId < STATE_COUNT))
for (Parent parent = stateParents[stateId];
parent;
parent = forkParent(parent.forkId))
		{
			HFSM2_ASSERT(parent.forkId != 0);

			if (parent.forkId > 0)
return parent.prong != compoActive	 [parent.forkId - 1] &&
parent.prong == compoRequested[parent.forkId - 1];
		}

	return false;
}

template <typename TG_, typename TSL_, typename TRL_, Long NCC_, Long NOC_, Long NOU_, typename TRO_ HFSM2_IF_SERIALIZATION(, Long NSB_) HFSM2_IF_PLANS(, Long NTC_), typename TTP_>
HFSM2_CONSTEXPR(14)
bool
RegistryT<ArgsT<TG_, TSL_, TRL_, NCC_, NOC_, NOU_, TRO_ HFSM2_IF_SERIALIZATION(, NSB_) HFSM2_IF_PLANS(, NTC_), TTP_>>::isPendingExit(const StateID stateId) const noexcept {
	if (HFSM2_CHECKED(stateId < STATE_COUNT))
for (Parent parent = stateParents[stateId];
parent;
parent = forkParent(parent.forkId))
		{
			HFSM2_ASSERT(parent.forkId != 0);

			if (parent.forkId > 0)
return parent.prong == compoActive	 [parent.forkId - 1] &&
parent.prong != compoRequested[parent.forkId - 1];
		}

	return false;
}

template <typename TG_, typename TSL_, typename TRL_, Long NCC_, Long NOC_, Long NOU_, typename TRO_ HFSM2_IF_SERIALIZATION(, Long NSB_) HFSM2_IF_PLANS(, Long NTC_), typename TTP_>
HFSM2_CONSTEXPR(14)
const Parent&
RegistryT<ArgsT<TG_, TSL_, TRL_, NCC_, NOC_, NOU_, TRO_ HFSM2_IF_SERIALIZATION(, NSB_) HFSM2_IF_PLANS(, NTC_), TTP_>>::forkParent(const ForkID forkId) const noexcept {
	HFSM2_ASSERT(forkId != 0);

	return forkId > 0 ?
compoParents[ forkId - 1] :
orthoParents[-forkId - 1];
}

template <typename TG_, typename TSL_, typename TRL_, Long NCC_, Long NOC_, Long NOU_, typename TRO_ HFSM2_IF_SERIALIZATION(, Long NSB_) HFSM2_IF_PLANS(, Long NTC_), typename TTP_>
HFSM2_CONSTEXPR(14)
typename RegistryT<ArgsT<TG_, TSL_, TRL_, NCC_, NOC_, NOU_, TRO_ HFSM2_IF_SERIALIZATION(, NSB_) HFSM2_IF_PLANS(, NTC_), TTP_>>::OrthoBits
RegistryT<ArgsT<TG_, TSL_, TRL_, NCC_, NOC_, NOU_, TRO_ HFSM2_IF_SERIALIZATION(, NSB_) HFSM2_IF_PLANS(, NTC_), TTP_>>::requestedOrthoFork(const ForkID forkId) noexcept {
	HFSM2_ASSERT(forkId < 0);
const Units& units = orthoUnits[-forkId - 1];

	return orthoRequested.bits(units);
}

template <typename TG_, typename TSL_, typename TRL_, Long NCC_, Long NOC_, Long NOU_, typename TRO_ HFSM2_IF_SERIALIZATION(, Long NSB_) HFSM2_IF_PLANS(, Long NTC_), typename TTP_>
HFSM2_CONSTEXPR(14)
bool
RegistryT<ArgsT<TG_, TSL_, TRL_, NCC_, NOC_, NOU_, TRO_ HFSM2_IF_SERIALIZATION(, NSB_) HFSM2_IF_PLANS(, NTC_), TTP_>>::requestImmediate(const Transition& request) noexcept {
	if (request.destination == 0)
		return false;
	else if (HFSM2_CHECKED(request.destination < STATE_COUNT)) {
Parent parent;

for (parent = stateParents[request.destination];
parent;
parent = forkParent(parent.forkId))
		{
			if (parent.forkId > 0) {
compoRequested[parent.forkId - 1] = parent.prong;
parent = forkParent(parent.forkId);

				break;
			} else if (parent.forkId < 0)
				requestedOrthoFork(parent.forkId).set(parent.prong);
			else
				HFSM2_BREAK();
		}

for (; parent; parent = forkParent(parent.forkId)) {
			if (parent.forkId > 0) {
				compoRemains.set(parent.forkId - 1);

if (compoActive	  [parent.forkId - 1] != parent.prong)
compoRequested[parent.forkId - 1]  = parent.prong;
				else {
parent = forkParent(parent.forkId);
					break;
				}
			} else if (parent.forkId < 0)
				requestedOrthoFork(parent.forkId).set(parent.prong);
			else
				HFSM2_BREAK();
		}

for (; parent; parent = forkParent(parent.forkId)) {
			if (parent.forkId > 0)
				compoRemains.set(parent.forkId - 1);
			else if (parent.forkId < 0)
				requestedOrthoFork(parent.forkId).set(parent.prong);
			else
				HFSM2_BREAK();
		}
	}

	return true;
}

template <typename TG_, typename TSL_, typename TRL_, Long NCC_, Long NOC_, Long NOU_, typename TRO_ HFSM2_IF_SERIALIZATION(, Long NSB_) HFSM2_IF_PLANS(, Long NTC_), typename TTP_>
HFSM2_CONSTEXPR(14)
void
RegistryT<ArgsT<TG_, TSL_, TRL_, NCC_, NOC_, NOU_, TRO_ HFSM2_IF_SERIALIZATION(, NSB_) HFSM2_IF_PLANS(, NTC_), TTP_>>::requestScheduled(const StateID stateId) noexcept {
	if (HFSM2_CHECKED(stateId < STATE_COUNT)) {
const Parent parent = stateParents[stateId];

		HFSM2_ASSERT(parent.forkId != 0);
		if (parent.forkId > 0)
compoResumable[parent.forkId - 1] = parent.prong;
	}
}

template <typename TG_, typename TSL_, typename TRL_, Long NCC_, Long NOC_, Long NOU_, typename TRO_ HFSM2_IF_SERIALIZATION(, Long NSB_) HFSM2_IF_PLANS(, Long NTC_), typename TTP_>
HFSM2_CONSTEXPR(14)
void
RegistryT<ArgsT<TG_, TSL_, TRL_, NCC_, NOC_, NOU_, TRO_ HFSM2_IF_SERIALIZATION(, NSB_) HFSM2_IF_PLANS(, NTC_), TTP_>>::clearRequests() noexcept {
	compoRequested.clear();
	orthoRequested.clear();
	compoRemains  .clear();
}

template <typename TG_, typename TSL_, typename TRL_, Long NCC_, Long NOC_, Long NOU_, typename TRO_ HFSM2_IF_SERIALIZATION(, Long NSB_) HFSM2_IF_PLANS(, Long NTC_), typename TTP_>
HFSM2_CONSTEXPR(14)
void
RegistryT<ArgsT<TG_, TSL_, TRL_, NCC_, NOC_, NOU_, TRO_ HFSM2_IF_SERIALIZATION(, NSB_) HFSM2_IF_PLANS(, NTC_), TTP_>>::clear() noexcept {
	clearRequests();

	compoActive	  .clear();
	compoResumable.clear();
}

template <typename TG_, typename TSL_, typename TRL_, Long NCC_, Long NOC_, Long NOU_, typename TRO_ HFSM2_IF_SERIALIZATION(, Long NSB_) HFSM2_IF_PLANS(, Long NTC_), typename TTP_>
HFSM2_CONSTEXPR(11)
bool
RegistryT<ArgsT<TG_, TSL_, TRL_, NCC_, NOC_, NOU_, TRO_ HFSM2_IF_SERIALIZATION(, NSB_) HFSM2_IF_PLANS(, NTC_), TTP_>>::empty() const noexcept {
	return compoRequested.empty()
		&& orthoRequested.empty()
		&& compoRemains	 .empty()
		&& compoActive	 .empty()
		&& compoResumable.empty();
}

}
}

namespace hfsm2 {
	namespace detail {

		template <typename TG_, typename TSL_, typename TRL_, Long NCC_, typename TRO_ HFSM2_IF_SERIALIZATION(, Long NSB_) HFSM2_IF_PLANS(, Long NTC_), typename TTP_>
		HFSM2_CONSTEXPR(14)
		Prong
		RegistryT<ArgsT<TG_, TSL_, TRL_, NCC_, 0, 0, TRO_ HFSM2_IF_SERIALIZATION(, NSB_) HFSM2_IF_PLANS(, NTC_), TTP_>>::activeSubState(const StateID stateId) const noexcept {
		const StateID subStateId = stateId + 1;

		if (HFSM2_CHECKED(	 stateId < STATE_COUNT) &&
		HFSM2_CHECKED(subStateId < STATE_COUNT))
		{
		if (const Parent parent = stateParents[subStateId]) {
		HFSM2_ASSERT(parent.forkId != 0);

		if (parent.forkId > 0)
		return compoActive[parent.forkId - 1];
	}
}

	return INVALID_PRONG;
}

template <typename TG_, typename TSL_, typename TRL_, Long NCC_, typename TRO_ HFSM2_IF_SERIALIZATION(, Long NSB_) HFSM2_IF_PLANS(, Long NTC_), typename TTP_>
HFSM2_CONSTEXPR(11)
bool
RegistryT<ArgsT<TG_, TSL_, TRL_, NCC_, 0, 0, TRO_ HFSM2_IF_SERIALIZATION(, NSB_) HFSM2_IF_PLANS(, NTC_), TTP_>>::isActive() const noexcept {
return compoActive[ROOT_ID] != INVALID_PRONG;
}

template <typename TG_, typename TSL_, typename TRL_, Long NCC_, typename TRO_ HFSM2_IF_SERIALIZATION(, Long NSB_) HFSM2_IF_PLANS(, Long NTC_), typename TTP_>
HFSM2_CONSTEXPR(14)
bool
RegistryT<ArgsT<TG_, TSL_, TRL_, NCC_, 0, 0, TRO_ HFSM2_IF_SERIALIZATION(, NSB_) HFSM2_IF_PLANS(, NTC_), TTP_>>::isActive(const StateID stateId) const noexcept {
	if (HFSM2_CHECKED(stateId < STATE_COUNT)) {
if (Parent parent = stateParents[stateId]) {
			HFSM2_ASSERT(parent.forkId > 0);

return parent.prong == compoActive[parent.forkId - 1];
		} else
			return isActive();
	}

	return false;
}

template <typename TG_, typename TSL_, typename TRL_, Long NCC_, typename TRO_ HFSM2_IF_SERIALIZATION(, Long NSB_) HFSM2_IF_PLANS(, Long NTC_), typename TTP_>
HFSM2_CONSTEXPR(14)
bool
RegistryT<ArgsT<TG_, TSL_, TRL_, NCC_, 0, 0, TRO_ HFSM2_IF_SERIALIZATION(, NSB_) HFSM2_IF_PLANS(, NTC_), TTP_>>::isResumable(const StateID stateId) const noexcept {
	if (HFSM2_CHECKED(stateId < STATE_COUNT))
if (Parent parent = stateParents[stateId]) {
			HFSM2_ASSERT(parent.forkId > 0);

return parent.prong == compoResumable[parent.forkId - 1];
		}

	return false;
}

template <typename TG_, typename TSL_, typename TRL_, Long NCC_, typename TRO_ HFSM2_IF_SERIALIZATION(, Long NSB_) HFSM2_IF_PLANS(, Long NTC_), typename TTP_>
HFSM2_CONSTEXPR(14)
bool
RegistryT<ArgsT<TG_, TSL_, TRL_, NCC_, 0, 0, TRO_ HFSM2_IF_SERIALIZATION(, NSB_) HFSM2_IF_PLANS(, NTC_), TTP_>>::isPendingChange(const StateID stateId) const noexcept {
	if (HFSM2_CHECKED(stateId < STATE_COUNT))
if (Parent parent = stateParents[stateId]) {
			HFSM2_ASSERT(parent.forkId > 0);

return compoRequested[parent.forkId - 1] !=
compoActive	 [parent.forkId - 1];
		}

	return false;
}

template <typename TG_, typename TSL_, typename TRL_, Long NCC_, typename TRO_ HFSM2_IF_SERIALIZATION(, Long NSB_) HFSM2_IF_PLANS(, Long NTC_), typename TTP_>
HFSM2_CONSTEXPR(14)
bool
RegistryT<ArgsT<TG_, TSL_, TRL_, NCC_, 0, 0, TRO_ HFSM2_IF_SERIALIZATION(, NSB_) HFSM2_IF_PLANS(, NTC_), TTP_>>::isPendingEnter(const StateID stateId) const noexcept {
	if (HFSM2_CHECKED(stateId < STATE_COUNT))
if (Parent parent = stateParents[stateId]) {
			HFSM2_ASSERT(parent.forkId > 0);

return parent.prong != compoActive	 [parent.forkId - 1] &&
parent.prong == compoRequested[parent.forkId - 1];
		}

	return false;
}

template <typename TG_, typename TSL_, typename TRL_, Long NCC_, typename TRO_ HFSM2_IF_SERIALIZATION(, Long NSB_) HFSM2_IF_PLANS(, Long NTC_), typename TTP_>
HFSM2_CONSTEXPR(14)
bool
RegistryT<ArgsT<TG_, TSL_, TRL_, NCC_, 0, 0, TRO_ HFSM2_IF_SERIALIZATION(, NSB_) HFSM2_IF_PLANS(, NTC_), TTP_>>::isPendingExit(const StateID stateId) const noexcept {
	if (HFSM2_CHECKED(stateId < STATE_COUNT))
if (Parent parent = stateParents[stateId]) {
			HFSM2_ASSERT(parent.forkId > 0);

return parent.prong == compoActive	 [parent.forkId - 1] &&
parent.prong != compoRequested[parent.forkId - 1];
		}

	return false;
}

template <typename TG_, typename TSL_, typename TRL_, Long NCC_, typename TRO_ HFSM2_IF_SERIALIZATION(, Long NSB_) HFSM2_IF_PLANS(, Long NTC_), typename TTP_>
HFSM2_CONSTEXPR(14)
const Parent&
RegistryT<ArgsT<TG_, TSL_, TRL_, NCC_, 0, 0, TRO_ HFSM2_IF_SERIALIZATION(, NSB_) HFSM2_IF_PLANS(, NTC_), TTP_>>::forkParent(const ForkID forkId) const noexcept {
	HFSM2_ASSERT(forkId > 0);

return compoParents[forkId - 1];
}

template <typename TG_, typename TSL_, typename TRL_, Long NCC_, typename TRO_ HFSM2_IF_SERIALIZATION(, Long NSB_) HFSM2_IF_PLANS(, Long NTC_), typename TTP_>
HFSM2_CONSTEXPR(14)
bool
RegistryT<ArgsT<TG_, TSL_, TRL_, NCC_, 0, 0, TRO_ HFSM2_IF_SERIALIZATION(, NSB_) HFSM2_IF_PLANS(, NTC_), TTP_>>::requestImmediate(const Transition& request) noexcept {
	// record request
	// promote it to all children
```
